    |   movel([0.360000, -1.280308, -2.635825, -0.796256, 1.570796, 1.930796],accel_mss,speed_ms,0,blend_radius_m)
    |   movel([0.360158, -1.281026, -2.635415, -0.795948, 1.570796, 1.930954],accel_mss,speed_ms,0,blend_radius_m)
    |   movel([0.360117, -1.282337, -2.634665, -0.795387, 1.570796, 1.930913],accel_mss,speed_ms,0,blend_radius_m)
    |   movel([0.359973, -1.283681, -2.633894, -0.794814, 1.570796, 1.930769],accel_mss,speed_ms,0,blend_radius_m)
    |   movel([0.359706, -1.284183, -2.633605, -0.794600, 1.570796, 1.930502],accel_mss,speed_ms,0,blend_radius_m)
    |   movel([0.359553, -1.284531, -2.633405, -0.794453, 1.570796, 1.930349],accel_mss,speed_ms,0,blend_radius_m)
    |   movel([0.359665, -1.284681, -2.633319, -0.794389, 1.570796, 1.930461],accel_mss,speed_ms,0,blend_radius_m)
    |   movel([0.360589, -1.285200, -2.633020, -0.794169, 1.570796, 1.931386],accel_mss,speed_ms,0,blend_radius_m)
    |   movel([0.360909, -1.283859, -2.633792, -0.794738, 1.570796, 1.931705],accel_mss,speed_ms,0,blend_radius_m)
    |   movel([0.361092, -1.281386, -2.635209, -0.795794, 1.570796, 1.931889],accel_mss,speed_ms,0,blend_radius_m)
    |   speed_ms = 0.005
    |   movel([0.361092, -1.272070, -2.630766, -0.809554, 1.570796, 1.931889],accel_mss,speed_ms,0,blend_radius_m)
    |   speed_ms = 0.040
    |   movel([0.352046, -1.270244, -2.631793, -0.810352, 1.570796, 1.922843],accel_mss,speed_ms,0,blend_radius_m)
    |   speed_ms = 0.005
    |   movel([0.352046, -1.279570, -2.636246, -0.796574, 1.570796, 1.922843],accel_mss,speed_ms,0,blend_radius_m)
    |   speed_ms = 0.025
    |   movel([0.350726, -1.280552, -2.635686, -0.796151, 1.570796, 1.921522],accel_mss,speed_ms,0,blend_radius_m)
    |   movel([0.350409, -1.280755, -2.635570, -0.796064, 1.570796, 1.921205],accel_mss,speed_ms,0,blend_radius_m)
    |   movel([0.349573, -1.281438, -2.635180, -0.795771, 1.570796, 1.920369],accel_mss,speed_ms,0,blend_radius_m)
    |   movel([0.349367, -1.281688, -2.635037, -0.795664, 1.570796, 1.920163],accel_mss,speed_ms,0,blend_radius_m)
    |   movel([0.349281, -1.282014, -2.634850, -0.795525, 1.570796, 1.920078],accel_mss,speed_ms,0,blend_radius_m)
    |   movel([0.349376, -1.282211, -2.634737, -0.795441, 1.570796, 1.920172],accel_mss,speed_ms,0,blend_radius_m)
    |   movel([0.349450, -1.282722, -2.634445, -0.795223, 1.570796, 1.920246],accel_mss,speed_ms,0,blend_radius_m)
    |   movel([0.349219, -1.283722, -2.633871, -0.794797, 1.570796, 1.920015],accel_mss,speed_ms,0,blend_radius_m)
    |   movel([0.348833, -1.284811, -2.633244, -0.794334, 1.570796, 1.919629],accel_mss,speed_ms,0,blend_radius_m)
    |   movel([0.348360, -1.285691, -2.632736, -0.793961, 1.570796, 1.919156],accel_mss,speed_ms,0,blend_radius_m)
    |   movel([0.346176, -1.288603, -2.631050, -0.792735, 1.570796, 1.916973],accel_mss,speed_ms,0,blend_radius_m)
    |   movel([0.345853, -1.288937, -2.630857, -0.792595, 1.570796, 1.916649],accel_mss,speed_ms,0,blend_radius_m)
    |   movel([0.345592, -1.289084, -2.630771, -0.792534, 1.570796, 1.916388],accel_mss,speed_ms,0,blend_radius_m)
    |   movel([0.345282, -1.289128, -2.630746, -0.792515, 1.570796, 1.916078],accel_mss,speed_ms,0,blend_radius_m)
    |   movel([0.344779, -1.289269, -2.630664, -0.792457, 1.570796, 1.915576],accel_mss,speed_ms,0,blend_radius_m)
    |   movel([0.344577, -1.289528, -2.630513, -0.792348, 1.570796, 1.915373],accel_mss,speed_ms,0,blend_radius_m)
    |   movel([0.343400, -1.291475, -2.629377, -0.791537, 1.570796, 1.914196],accel_mss,speed_ms,0,blend_radius_m)
    |   movel([0.342359, -1.292811, -2.628595, -0.790983, 1.570796, 1.913155],accel_mss,speed_ms,0,blend_radius_m)
    |   movel([0.341234, -1.294031, -2.627879, -0.790479, 1.570796, 1.912031],accel_mss,speed_ms,0,blend_radius_m)
    |   movel([0.340185, -1.294941, -2.627344, -0.790104, 1.570796, 1.910981],accel_mss,speed_ms,0,blend_radius_m)
    |   movel([0.339211, -1.295614, -2.626947, -0.789828, 1.570796, 1.910007],accel_mss,speed_ms,0,blend_radius_m)
    |   movel([0.338682, -1.295791, -2.626843, -0.789755, 1.570796, 1.909478],accel_mss,speed_ms,0,blend_radius_m)
    |   movel([0.338447, -1.295587, -2.626963, -0.789839, 1.570796, 1.909243],accel_mss,speed_ms,0,blend_radius_m)
    |   movel([0.338512, -1.294948, -2.627340, -0.790101, 1.570796, 1.909309],accel_mss,speed_ms,0,blend_radius_m)
    |   movel([0.338713, -1.294120, -2.627827, -0.790442, 1.570796, 1.909510],accel_mss,speed_ms,0,blend_radius_m)
    |   movel([0.338129, -1.294814, -2.627419, -0.790156, 1.570796, 1.908925],accel_mss,speed_ms,0,blend_radius_m)
    |   movel([0.335286, -1.297812, -2.625648, -0.788929, 1.570796, 1.906082],accel_mss,speed_ms,0,blend_radius_m)
    |   movel([0.333596, -1.299421, -2.624693, -0.788275, 1.570796, 1.904392],accel_mss,speed_ms,0,blend_radius_m)
    |   movel([0.330932, -1.301652, -2.623363, -0.787375, 1.570796, 1.901728],accel_mss,speed_ms,0,blend_radius_m)
    |   movel([0.330138, -1.302174, -2.623051, -0.787165, 1.570796, 1.900934],accel_mss,speed_ms,0,blend_radius_m)
    |   movel([0.329651, -1.302339, -2.622952, -0.787098, 1.570796, 1.900448],accel_mss,speed_ms,0,blend_radius_m)
    |   movel([0.329404, -1.302208, -2.623030, -0.787151, 1.570796, 1.900200],accel_mss,speed_ms,0,blend_radius_m)
    |   movel([0.329712, -1.301575, -2.623409, -0.787406, 1.570796, 1.900508],accel_mss,speed_ms,0,blend_radius_m)
    |   movel([0.330081, -1.300968, -2.623771, -0.787650, 1.570796, 1.900877],accel_mss,speed_ms,0,blend_radius_m)
    |   movel([0.331306, -1.299082, -2.624894, -0.788413, 1.570796, 1.902102],accel_mss,speed_ms,0,blend_radius_m)
    |   movel([0.331670, -1.298377, -2.625312, -0.788699, 1.570796, 1.902467],accel_mss,speed_ms,0,blend_radius_m)
    |   movel([0.332580, -1.295268, -2.627151, -0.789970, 1.570796, 1.903377],accel_mss,speed_ms,0,blend_radius_m)
    |   movel([0.332687, -1.295094, -2.627254, -0.790041, 1.570796, 1.903483],accel_mss,speed_ms,0,blend_radius_m)
    |   movel([0.333051, -1.294898, -2.627369, -0.790122, 1.570796, 1.903847],accel_mss,speed_ms,0,blend_radius_m)
    |   movel([0.333400, -1.294997, -2.627311, -0.790081, 1.570796, 1.904196],accel_mss,speed_ms,0,blend_radius_m)
    |   movel([0.333513, -1.295473, -2.627031, -0.789886, 1.570796, 1.904310],accel_mss,speed_ms,0,blend_radius_m)
    |   movel([0.333369, -1.296352, -2.626512, -0.789526, 1.570796, 1.904165],accel_mss,speed_ms,0,blend_radius_m)
    |   movel([0.332468, -1.299246, -2.624796, -0.788346, 1.570796, 1.903264],accel_mss,speed_ms,0,blend_radius_m)
    |   movel([0.333060, -1.298841, -2.625038, -0.788511, 1.570796, 1.903857],accel_mss,speed_ms,0,blend_radius_m)
    |   movel([0.334701, -1.297178, -2.626023, -0.789188, 1.570796, 1.905498],accel_mss,speed_ms,0,blend_radius_m)
    |   movel([0.339129, -1.292381, -2.628847, -0.791161, 1.570796, 1.909925],accel_mss,speed_ms,0,blend_radius_m)
    |   movel([0.339470, -1.292099, -2.629012, -0.791278, 1.570796, 1.910266],accel_mss,speed_ms,0,blend_radius_m)
    |   movel([0.339852, -1.291915, -2.629120, -0.791354, 1.570796, 1.910648],accel_mss,speed_ms,0,blend_radius_m)
    |   movel([0.340105, -1.291922, -2.629116, -0.791351, 1.570796, 1.910901],accel_mss,speed_ms,0,blend_radius_m)
    |   movel([0.340213, -1.292101, -2.629011, -0.791277, 1.570796, 1.911009],accel_mss,speed_ms,0,blend_radius_m)
    |   movel([0.340131, -1.293204, -2.628365, -0.790820, 1.570796, 1.910927],accel_mss,speed_ms,0,blend_radius_m)
    |   movel([0.340095, -1.293842, -2.627990, -0.790557, 1.570796, 1.910891],accel_mss,speed_ms,0,blend_radius_m)
    |   movel([0.340385, -1.293737, -2.628052, -0.790600, 1.570796, 1.911181],accel_mss,speed_ms,0,blend_radius_m)
    |   movel([0.341029, -1.293046, -2.628457, -0.790885, 1.570796, 1.911825],accel_mss,speed_ms,0,blend_radius_m)
    |   movel([0.342320, -1.291451, -2.629392, -0.791547, 1.570796, 1.913117],accel_mss,speed_ms,0,blend_radius_m)
    |   movel([0.342678, -1.290913, -2.629706, -0.791771, 1.570796, 1.913474],accel_mss,speed_ms,0,blend_radius_m)
    |   movel([0.344707, -1.287200, -2.631864, -0.793325, 1.570796, 1.915504],accel_mss,speed_ms,0,blend_radius_m)
    |   movel([0.345022, -1.286686, -2.632162, -0.793541, 1.570796, 1.915819],accel_mss,speed_ms,0,blend_radius_m)
    |   movel([0.345276, -1.286420, -2.632316, -0.793654, 1.570796, 1.916072],accel_mss,speed_ms,0,blend_radius_m)
    |   movel([0.345565, -1.286274, -2.632400, -0.793715, 1.570796, 1.916361],accel_mss,speed_ms,0,blend_radius_m)
    |   movel([0.345919, -1.286308, -2.632380, -0.793701, 1.570796, 1.916715],accel_mss,speed_ms,0,blend_radius_m)
    |   movel([0.345989, -1.286458, -2.632294, -0.793638, 1.570796, 1.916786],accel_mss,speed_ms,0,blend_radius_m)
    |   movel([0.346060, -1.287092, -2.631927, -0.793370, 1.570796, 1.916857],accel_mss,speed_ms,0,blend_radius_m)
    |   movel([0.346199, -1.287137, -2.631901, -0.793351, 1.570796, 1.916995],accel_mss,speed_ms,0,blend_radius_m)
    |   movel([0.346613, -1.286673, -2.632169, -0.793547, 1.570796, 1.917409],accel_mss,speed_ms,0,blend_radius_m)
    |   movel([0.347721, -1.284766, -2.633270, -0.794353, 1.570796, 1.918517],accel_mss,speed_ms,0,blend_radius_m)
    |   movel([0.348015, -1.284034, -2.633691, -0.794664, 1.570796, 1.918811],accel_mss,speed_ms,0,blend_radius_m)
    |   movel([0.348173, -1.283275, -2.634127, -0.794987, 1.570796, 1.918969],accel_mss,speed_ms,0,blend_radius_m)
    |   movel([0.348061, -1.283203, -2.634169, -0.795018, 1.570796, 1.918858],accel_mss,speed_ms,0,blend_radius_m)
    |   movel([0.347358, -1.283201, -2.634170, -0.795018, 1.570796, 1.918154],accel_mss,speed_ms,0,blend_radius_m)
    |   movel([0.347299, -1.282914, -2.634334, -0.795141, 1.570796, 1.918095],accel_mss,speed_ms,0,blend_radius_m)
    |   movel([0.347686, -1.282282, -2.634697, -0.795411, 1.570796, 1.918482],accel_mss,speed_ms,0,blend_radius_m)
    |   movel([0.348658, -1.281144, -2.635348, -0.795897, 1.570796, 1.919454],accel_mss,speed_ms,0,blend_radius_m)
    |   movel([0.350016, -1.279729, -2.636155, -0.796505, 1.570796, 1.920812],accel_mss,speed_ms,0,blend_radius_m)
    |   movel([0.350378, -1.279523, -2.636273, -0.796594, 1.570796, 1.921174],accel_mss,speed_ms,0,blend_radius_m)
    |   movel([0.351006, -1.279344, -2.636374, -0.796671, 1.570796, 1.921802],accel_mss,speed_ms,0,blend_radius_m)
    |   movel([0.351161, -1.279219, -2.636445, -0.796725, 1.570796, 1.921958],accel_mss,speed_ms,0,blend_radius_m)
    |   movel([0.351485, -1.278767, -2.636702, -0.796920, 1.570796, 1.922281],accel_mss,speed_ms,0,blend_radius_m)
    |   movel([0.351478, -1.278534, -2.636835, -0.797020, 1.570796, 1.922274],accel_mss,speed_ms,0,blend_radius_m)
    |   movel([0.350699, -1.278105, -2.637078, -0.797206, 1.570796, 1.921496],accel_mss,speed_ms,0,blend_radius_m)
    |   movel([0.350151, -1.277985, -2.637146, -0.797258, 1.570796, 1.920947],accel_mss,speed_ms,0,blend_radius_m)
    |   movel([0.348867, -1.278148, -2.637054, -0.797187, 1.570796, 1.919663],accel_mss,speed_ms,0,blend_radius_m)
    |   movel([0.348187, -1.278424, -2.636897, -0.797068, 1.570796, 1.918984],accel_mss,speed_ms,0,blend_radius_m)
    |   movel([0.346556, -1.279452, -2.636312, -0.796624, 1.570796, 1.917352],accel_mss,speed_ms,0,blend_radius_m)
    |   movel([0.344489, -1.281187, -2.635323, -0.795879, 1.570796, 1.915285],accel_mss,speed_ms,0,blend_radius_m)
    |   movel([0.342140, -1.283410, -2.634050, -0.794929, 1.570796, 1.912937],accel_mss,speed_ms,0,blend_radius_m)
    |   movel([0.339990, -1.285647, -2.632762, -0.793980, 1.570796, 1.910786],accel_mss,speed_ms,0,blend_radius_m)
    |   movel([0.338281, -1.287605, -2.631630, -0.793154, 1.570796, 1.909077],accel_mss,speed_ms,0,blend_radius_m)
    |   movel([0.337925, -1.288106, -2.631339, -0.792944, 1.570796, 1.908722],accel_mss,speed_ms,0,blend_radius_m)
    |   movel([0.337295, -1.289450, -2.630558, -0.792381, 1.570796, 1.908092],accel_mss,speed_ms,0,blend_radius_m)
    |   movel([0.336751, -1.290223, -2.630108, -0.792058, 1.570796, 1.907547],accel_mss,speed_ms,0,blend_radius_m)
    |   movel([0.335966, -1.291041, -2.629631, -0.791717, 1.570796, 1.906762],accel_mss,speed_ms,0,blend_radius_m)
    |   movel([0.334835, -1.292017, -2.629060, -0.791312, 1.570796, 1.905631],accel_mss,speed_ms,0,blend_radius_m)
    |   movel([0.333094, -1.293432, -2.628231, -0.790726, 1.570796, 1.903890],accel_mss,speed_ms,0,blend_radius_m)
    |   movel([0.333989, -1.293324, -2.628294, -0.790771, 1.570796, 1.904785],accel_mss,speed_ms,0,blend_radius_m)
    |   movel([0.334947, -1.293151, -2.628396, -0.790842, 1.570796, 1.905743],accel_mss,speed_ms,0,blend_radius_m)
    |   movel([0.335825, -1.292864, -2.628564, -0.790961, 1.570796, 1.906621],accel_mss,speed_ms,0,blend_radius_m)
    |   movel([0.336611, -1.292469, -2.628796, -0.791124, 1.570796, 1.907408],accel_mss,speed_ms,0,blend_radius_m)
    |   movel([0.337314, -1.291964, -2.629091, -0.791334, 1.570796, 1.908110],accel_mss,speed_ms,0,blend_radius_m)
    |   movel([0.339476, -1.289654, -2.630440, -0.792296, 1.570796, 1.910272],accel_mss,speed_ms,0,blend_radius_m)
    |   movel([0.340428, -1.288554, -2.631079, -0.792756, 1.570796, 1.911224],accel_mss,speed_ms,0,blend_radius_m)
    |   movel([0.342358, -1.286351, -2.632355, -0.793683, 1.570796, 1.913154],accel_mss,speed_ms,0,blend_radius_m)
    |   movel([0.343884, -1.284770, -2.633268, -0.794351, 1.570796, 1.914681],accel_mss,speed_ms,0,blend_radius_m)
    |   movel([0.345057, -1.283720, -2.633872, -0.794798, 1.570796, 1.915853],accel_mss,speed_ms,0,blend_radius_m)
    |   movel([0.345391, -1.283506, -2.633994, -0.794888, 1.570796, 1.916188],accel_mss,speed_ms,0,blend_radius_m)
    |   movel([0.345733, -1.283407, -2.634051, -0.794931, 1.570796, 1.916529],accel_mss,speed_ms,0,blend_radius_m)
    |   movel([0.346062, -1.283485, -2.634007, -0.794897, 1.570796, 1.916858],accel_mss,speed_ms,0,blend_radius_m)
    |   movel([0.346078, -1.283751, -2.633854, -0.794784, 1.570796, 1.916875],accel_mss,speed_ms,0,blend_radius_m)
    |   movel([0.345707, -1.284258, -2.633562, -0.794569, 1.570796, 1.916503],accel_mss,speed_ms,0,blend_radius_m)
    |   movel([0.343367, -1.286602, -2.632210, -0.793577, 1.570796, 1.914163],accel_mss,speed_ms,0,blend_radius_m)
    |   movel([0.342356, -1.287721, -2.631562, -0.793106, 1.570796, 1.913152],accel_mss,speed_ms,0,blend_radius_m)
    |   movel([0.339475, -1.291018, -2.629644, -0.791727, 1.570796, 1.910271],accel_mss,speed_ms,0,blend_radius_m)
    |   movel([0.338056, -1.292411, -2.628830, -0.791148, 1.570796, 1.908853],accel_mss,speed_ms,0,blend_radius_m)
    |   movel([0.336846, -1.293317, -2.628299, -0.790774, 1.570796, 1.907642],accel_mss,speed_ms,0,blend_radius_m)
    |   movel([0.335632, -1.293912, -2.627949, -0.790528, 1.570796, 1.906428],accel_mss,speed_ms,0,blend_radius_m)
    |   movel([0.332841, -1.294566, -2.627564, -0.790258, 1.570796, 1.903637],accel_mss,speed_ms,0,blend_radius_m)
    |   movel([0.331679, -1.294769, -2.627445, -0.790175, 1.570796, 1.902475],accel_mss,speed_ms,0,blend_radius_m)
    |   movel([0.329311, -1.295109, -2.627245, -0.790035, 1.570796, 1.900107],accel_mss,speed_ms,0,blend_radius_m)
    |   movel([0.328965, -1.295079, -2.627263, -0.790048, 1.570796, 1.899762],accel_mss,speed_ms,0,blend_radius_m)
    |   movel([0.328847, -1.294931, -2.627350, -0.790108, 1.570796, 1.899643],accel_mss,speed_ms,0,blend_radius_m)
    |   movel([0.328941, -1.294638, -2.627522, -0.790229, 1.570796, 1.899737],accel_mss,speed_ms,0,blend_radius_m)
    |   movel([0.329215, -1.294351, -2.627691, -0.790347, 1.570796, 1.900011],accel_mss,speed_ms,0,blend_radius_m)
    |   movel([0.329727, -1.294034, -2.627877, -0.790478, 1.570796, 1.900523],accel_mss,speed_ms,0,blend_radius_m)
    |   movel([0.331665, -1.293098, -2.628427, -0.790864, 1.570796, 1.902462],accel_mss,speed_ms,0,blend_radius_m)
    |   movel([0.332996, -1.292293, -2.628899, -0.791197, 1.570796, 1.903793],accel_mss,speed_ms,0,blend_radius_m)
    |   movel([0.334270, -1.291420, -2.629410, -0.791560, 1.570796, 1.905066],accel_mss,speed_ms,0,blend_radius_m)
    |   movel([0.335177, -1.290667, -2.629849, -0.791873, 1.570796, 1.905974],accel_mss,speed_ms,0,blend_radius_m)
    |   movel([0.335919, -1.289820, -2.630343, -0.792226, 1.570796, 1.906715],accel_mss,speed_ms,0,blend_radius_m)
    |   movel([0.336246, -1.289316, -2.630636, -0.792437, 1.570796, 1.907043],accel_mss,speed_ms,0,blend_radius_m)
    |   movel([0.337469, -1.287167, -2.631884, -0.793339, 1.570796, 1.908266],accel_mss,speed_ms,0,blend_radius_m)
    |   movel([0.337607, -1.286986, -2.631988, -0.793415, 1.570796, 1.908403],accel_mss,speed_ms,0,blend_radius_m)
    |   movel([0.337528, -1.286900, -2.632038, -0.793451, 1.570796, 1.908324],accel_mss,speed_ms,0,blend_radius_m)
    |   movel([0.337263, -1.286966, -2.632000, -0.793423, 1.570796, 1.908059],accel_mss,speed_ms,0,blend_radius_m)
    |   movel([0.336794, -1.286946, -2.632011, -0.793432, 1.570796, 1.907591],accel_mss,speed_ms,0,blend_radius_m)
    |   movel([0.336758, -1.286839, -2.632073, -0.793477, 1.570796, 1.907555],accel_mss,speed_ms,0,blend_radius_m)
    |   movel([0.336882, -1.286488, -2.632276, -0.793625, 1.570796, 1.907678],accel_mss,speed_ms,0,blend_radius_m)
    |   movel([0.337579, -1.285557, -2.632814, -0.794018, 1.570796, 1.908376],accel_mss,speed_ms,0,blend_radius_m)
    |   movel([0.340525, -1.282052, -2.634828, -0.795509, 1.570796, 1.911322],accel_mss,speed_ms,0,blend_radius_m)
    |   movel([0.340661, -1.281806, -2.634969, -0.795614, 1.570796, 1.911457],accel_mss,speed_ms,0,blend_radius_m)
    |   movel([0.340523, -1.281433, -2.635183, -0.795774, 1.570796, 1.911319],accel_mss,speed_ms,0,blend_radius_m)
    |   movel([0.340591, -1.280649, -2.635631, -0.796110, 1.570796, 1.911388],accel_mss,speed_ms,0,blend_radius_m)
    |   movel([0.340729, -1.279843, -2.636090, -0.796456, 1.570796, 1.911526],accel_mss,speed_ms,0,blend_radius_m)
    |   movel([0.340926, -1.279484, -2.636294, -0.796610, 1.570796, 1.911722],accel_mss,speed_ms,0,blend_radius_m)
    |   movel([0.341239, -1.279281, -2.636410, -0.796698, 1.570796, 1.912035],accel_mss,speed_ms,0,blend_radius_m)
    |   movel([0.341530, -1.279306, -2.636396, -0.796687, 1.570796, 1.912326],accel_mss,speed_ms,0,blend_radius_m)
    |   movel([0.341737, -1.279581, -2.636239, -0.796569, 1.570796, 1.912533],accel_mss,speed_ms,0,blend_radius_m)
    |   movel([0.341803, -1.280049, -2.635973, -0.796368, 1.570796, 1.912599],accel_mss,speed_ms,0,blend_radius_m)
    |   movel([0.341795, -1.280796, -2.635547, -0.796047, 1.570796, 1.912592],accel_mss,speed_ms,0,blend_radius_m)
    |   movel([0.343174, -1.279535, -2.636265, -0.796588, 1.570796, 1.913971],accel_mss,speed_ms,0,blend_radius_m)
    |   movel([0.346049, -1.276916, -2.637752, -0.797721, 1.570796, 1.916846],accel_mss,speed_ms,0,blend_radius_m)
    |   movel([0.345679, -1.276653, -2.637901, -0.797835, 1.570796, 1.916476],accel_mss,speed_ms,0,blend_radius_m)
    |   movel([0.345163, -1.276545, -2.637962, -0.797882, 1.570796, 1.915960],accel_mss,speed_ms,0,blend_radius_m)
    |   movel([0.344787, -1.276712, -2.637868, -0.797809, 1.570796, 1.915584],accel_mss,speed_ms,0,blend_radius_m)
    |   movel([0.341919, -1.278507, -2.636850, -0.797032, 1.570796, 1.912716],accel_mss,speed_ms,0,blend_radius_m)
    |   movel([0.340652, -1.279583, -2.636238, -0.796568, 1.570796, 1.911449],accel_mss,speed_ms,0,blend_radius_m)
    |   movel([0.339694, -1.280798, -2.635545, -0.796046, 1.570796, 1.910490],accel_mss,speed_ms,0,blend_radius_m)
    |   movel([0.338762, -1.282492, -2.634576, -0.795321, 1.570796, 1.909558],accel_mss,speed_ms,0,blend_radius_m)
    |   movel([0.337668, -1.284650, -2.633337, -0.794402, 1.570796, 1.908464],accel_mss,speed_ms,0,blend_radius_m)
    |   movel([0.337414, -1.284913, -2.633185, -0.794291, 1.570796, 1.908211],accel_mss,speed_ms,0,blend_radius_m)
    |   movel([0.337121, -1.285037, -2.633114, -0.794238, 1.570796, 1.907917],accel_mss,speed_ms,0,blend_radius_m)
    |   movel([0.336837, -1.284954, -2.633162, -0.794273, 1.570796, 1.907633],accel_mss,speed_ms,0,blend_radius_m)
    |   movel([0.336775, -1.284660, -2.633331, -0.794398, 1.570796, 1.907571],accel_mss,speed_ms,0,blend_radius_m)
    |   movel([0.336965, -1.284046, -2.633684, -0.794659, 1.570796, 1.907762],accel_mss,speed_ms,0,blend_radius_m)
    |   movel([0.338700, -1.280649, -2.635630, -0.796110, 1.570796, 1.909496],accel_mss,speed_ms,0,blend_radius_m)
    |   movel([0.339219, -1.279877, -2.636071, -0.796441, 1.570796, 1.910015],accel_mss,speed_ms,0,blend_radius_m)
    |   movel([0.340505, -1.278475, -2.636868, -0.797046, 1.570796, 1.911301],accel_mss,speed_ms,0,blend_radius_m)
    |   movel([0.341242, -1.277887, -2.637202, -0.797300, 1.570796, 1.912038],accel_mss,speed_ms,0,blend_radius_m)
    |   movel([0.344850, -1.275621, -2.638484, -0.798284, 1.570796, 1.915646],accel_mss,speed_ms,0,blend_radius_m)
    |   movel([0.344975, -1.275480, -2.638564, -0.798345, 1.570796, 1.915771],accel_mss,speed_ms,0,blend_radius_m)
    |   movel([0.344967, -1.275345, -2.638640, -0.798404, 1.570796, 1.915763],accel_mss,speed_ms,0,blend_radius_m)
    |   movel([0.344595, -1.275334, -2.638646, -0.798409, 1.570796, 1.915392],accel_mss,speed_ms,0,blend_radius_m)
    |   movel([0.342920, -1.276167, -2.638176, -0.798046, 1.570796, 1.913716],accel_mss,speed_ms,0,blend_radius_m)
    |   movel([0.340911, -1.277359, -2.637501, -0.797528, 1.570796, 1.911707],accel_mss,speed_ms,0,blend_radius_m)
    |   movel([0.340160, -1.277929, -2.637178, -0.797282, 1.570796, 1.910956],accel_mss,speed_ms,0,blend_radius_m)
    |   movel([0.339476, -1.278577, -2.636810, -0.797002, 1.570796, 1.910272],accel_mss,speed_ms,0,blend_radius_m)
    |   movel([0.338291, -1.280119, -2.635933, -0.796337, 1.570796, 1.909087],accel_mss,speed_ms,0,blend_radius_m)
    |   movel([0.337053, -1.282368, -2.634647, -0.795373, 1.570796, 1.907849],accel_mss,speed_ms,0,blend_radius_m)
    |   movel([0.335830, -1.284771, -2.633267, -0.794351, 1.570796, 1.906627],accel_mss,speed_ms,0,blend_radius_m)
    |   movel([0.335570, -1.285106, -2.633074, -0.794209, 1.570796, 1.906366],accel_mss,speed_ms,0,blend_radius_m)
    |   movel([0.335251, -1.285332, -2.632944, -0.794113, 1.570796, 1.906047],accel_mss,speed_ms,0,blend_radius_m)
    |   movel([0.334956, -1.285396, -2.632907, -0.794086, 1.570796, 1.905752],accel_mss,speed_ms,0,blend_radius_m)
    |   movel([0.334753, -1.285283, -2.632972, -0.794134, 1.570796, 1.905550],accel_mss,speed_ms,0,blend_radius_m)
    |   movel([0.334737, -1.285068, -2.633096, -0.794225, 1.570796, 1.905533],accel_mss,speed_ms,0,blend_radius_m)
    |   movel([0.335255, -1.283844, -2.633800, -0.794745, 1.570796, 1.906051],accel_mss,speed_ms,0,blend_radius_m)
    |   movel([0.335912, -1.282552, -2.634542, -0.795295, 1.570796, 1.906709],accel_mss,speed_ms,0,blend_radius_m)
    |   movel([0.337597, -1.279500, -2.636285, -0.796603, 1.570796, 1.908393],accel_mss,speed_ms,0,blend_radius_m)
    |   movel([0.338195, -1.278676, -2.636754, -0.796959, 1.570796, 1.908991],accel_mss,speed_ms,0,blend_radius_m)
    |   movel([0.339703, -1.277153, -2.637618, -0.797618, 1.570796, 1.910499],accel_mss,speed_ms,0,blend_radius_m)
    |   movel([0.340471, -1.276557, -2.637955, -0.797876, 1.570796, 1.911267],accel_mss,speed_ms,0,blend_radius_m)
    |   movel([0.342715, -1.275234, -2.638703, -0.798452, 1.570796, 1.913511],accel_mss,speed_ms,0,blend_radius_m)
    |   movel([0.344071, -1.274571, -2.639076, -0.798742, 1.570796, 1.914867],accel_mss,speed_ms,0,blend_radius_m)
    |   movel([0.345029, -1.274259, -2.639252, -0.798878, 1.570796, 1.915825],accel_mss,speed_ms,0,blend_radius_m)
    |   movel([0.345612, -1.274279, -2.639241, -0.798869, 1.570796, 1.916408],accel_mss,speed_ms,0,blend_radius_m)
    |   movel([0.346261, -1.275264, -2.638686, -0.798439, 1.570796, 1.917057],accel_mss,speed_ms,0,blend_radius_m)
    |   movel([0.346498, -1.275497, -2.638554, -0.798338, 1.570796, 1.917295],accel_mss,speed_ms,0,blend_radius_m)
    |   movel([0.347072, -1.275880, -2.638338, -0.798171, 1.570796, 1.917869],accel_mss,speed_ms,0,blend_radius_m)
    |   movel([0.347297, -1.275882, -2.638337, -0.798170, 1.570796, 1.918094],accel_mss,speed_ms,0,blend_radius_m)
    |   movel([0.348230, -1.275526, -2.638538, -0.798325, 1.570796, 1.919027],accel_mss,speed_ms,0,blend_radius_m)
    |   movel([0.348990, -1.275437, -2.638588, -0.798364, 1.570796, 1.919786],accel_mss,speed_ms,0,blend_radius_m)
    |   movel([0.349669, -1.275526, -2.638538, -0.798325, 1.570796, 1.920466],accel_mss,speed_ms,0,blend_radius_m)
    |   movel([0.350116, -1.275789, -2.638390, -0.798211, 1.570796, 1.920912],accel_mss,speed_ms,0,blend_radius_m)
    |   movel([0.350438, -1.276356, -2.638069, -0.797964, 1.570796, 1.921235],accel_mss,speed_ms,0,blend_radius_m)
    |   movel([0.350427, -1.276487, -2.637995, -0.797907, 1.570796, 1.921223],accel_mss,speed_ms,0,blend_radius_m)
    |   movel([0.350632, -1.276776, -2.637832, -0.797782, 1.570796, 1.921429],accel_mss,speed_ms,0,blend_radius_m)
    |   movel([0.350810, -1.276823, -2.637805, -0.797761, 1.570796, 1.921606],accel_mss,speed_ms,0,blend_radius_m)
    |   movel([0.351648, -1.277063, -2.637669, -0.797657, 1.570796, 1.922445],accel_mss,speed_ms,0,blend_radius_m)
    |   movel([0.352340, -1.277521, -2.637409, -0.797458, 1.570796, 1.923136],accel_mss,speed_ms,0,blend_radius_m)
    |   movel([0.352766, -1.278081, -2.637092, -0.797216, 1.570796, 1.923562],accel_mss,speed_ms,0,blend_radius_m)
    |   movel([0.352762, -1.278621, -2.636785, -0.796983, 1.570796, 1.923559],accel_mss,speed_ms,0,blend_radius_m)
    |   movel([0.352273, -1.279335, -2.636379, -0.796675, 1.570796, 1.923069],accel_mss,speed_ms,0,blend_radius_m)
    |   movel([0.352046, -1.279570, -2.636246, -0.796574, 1.570796, 1.922843],accel_mss,speed_ms,0,blend_radius_m)
    |   movel([0.350726, -1.280552, -2.635686, -0.796151, 1.570796, 1.921522],accel_mss,speed_ms,0,blend_radius_m)
    |   movel([0.350409, -1.280755, -2.635570, -0.796064, 1.570796, 1.921205],accel_mss,speed_ms,0,blend_radius_m)
    |   movel([0.349573, -1.281438, -2.635180, -0.795771, 1.570796, 1.920369],accel_mss,speed_ms,0,blend_radius_m)
    |   movel([0.349449, -1.281590, -2.635093, -0.795706, 1.570796, 1.920245],accel_mss,speed_ms,0,blend_radius_m)
    |   speed_ms = 0.005
    |   movel([0.349449, -1.272274, -2.630650, -0.809465, 1.570796, 1.920245],accel_mss,speed_ms,0,blend_radius_m)
    |   speed_ms = 0.040
    |   movel([0.349144, -1.267306, -2.633439, -0.811644, 1.570796, 1.919941],accel_mss,speed_ms,0,blend_radius_m)
    |   speed_ms = 0.005
    |   movel([0.349144, -1.276648, -2.637904, -0.797837, 1.570796, 1.919941],accel_mss,speed_ms,0,blend_radius_m)
    |   speed_ms = 0.025
    |   movel([0.349180, -1.276811, -2.637812, -0.797766, 1.570796, 1.919976],accel_mss,speed_ms,0,blend_radius_m)
    |   movel([0.349084, -1.276963, -2.637725, -0.797700, 1.570796, 1.919880],accel_mss,speed_ms,0,blend_radius_m)
    |   movel([0.348249, -1.277348, -2.637508, -0.797533, 1.570796, 1.919045],accel_mss,speed_ms,0,blend_radius_m)
    |   movel([0.347099, -1.277982, -2.637148, -0.797259, 1.570796, 1.917896],accel_mss,speed_ms,0,blend_radius_m)
    |   movel([0.345154, -1.279499, -2.636286, -0.796604, 1.570796, 1.915950],accel_mss,speed_ms,0,blend_radius_m)
    |   movel([0.343016, -1.281354, -2.635228, -0.795807, 1.570796, 1.913812],accel_mss,speed_ms,0,blend_radius_m)
    |   movel([0.339384, -1.284965, -2.633155, -0.794269, 1.570796, 1.910180],accel_mss,speed_ms,0,blend_radius_m)
    |   movel([0.338860, -1.285472, -2.632863, -0.794054, 1.570796, 1.909657],accel_mss,speed_ms,0,blend_radius_m)
    |   movel([0.339303, -1.284870, -2.633210, -0.794309, 1.570796, 1.910099],accel_mss,speed_ms,0,blend_radius_m)
    |   movel([0.341971, -1.281947, -2.634889, -0.795554, 1.570796, 1.912767],accel_mss,speed_ms,0,blend_radius_m)
    |   movel([0.343425, -1.280525, -2.635701, -0.796163, 1.570796, 1.914221],accel_mss,speed_ms,0,blend_radius_m)
    |   movel([0.346674, -1.277583, -2.637374, -0.797432, 1.570796, 1.917470],accel_mss,speed_ms,0,blend_radius_m)
    |   movel([0.347380, -1.277019, -2.637694, -0.797676, 1.570796, 1.918176],accel_mss,speed_ms,0,blend_radius_m)
    |   movel([0.347867, -1.276745, -2.637849, -0.797795, 1.570796, 1.918663],accel_mss,speed_ms,0,blend_radius_m)
    |   movel([0.348359, -1.276612, -2.637924, -0.797853, 1.570796, 1.919155],accel_mss,speed_ms,0,blend_radius_m)
    |   movel([0.349144, -1.276648, -2.637904, -0.797837, 1.570796, 1.919941],accel_mss,speed_ms,0,blend_radius_m)
    |   movel([0.349180, -1.276811, -2.637812, -0.797766, 1.570796, 1.919976],accel_mss,speed_ms,0,blend_radius_m)
    |   movel([0.349084, -1.276963, -2.637725, -0.797700, 1.570796, 1.919880],accel_mss,speed_ms,0,blend_radius_m)
    |   movel([0.348249, -1.277348, -2.637508, -0.797533, 1.570796, 1.919045],accel_mss,speed_ms,0,blend_radius_m)
    |   movel([0.347099, -1.277982, -2.637148, -0.797259, 1.570796, 1.917896],accel_mss,speed_ms,0,blend_radius_m)
    |   movel([0.346664, -1.278321, -2.636955, -0.797112, 1.570796, 1.917460],accel_mss,speed_ms,0,blend_radius_m)
    |   speed_ms = 0.005
    |   movel([0.346664, -1.268989, -2.632498, -0.810902, 1.570796, 1.917460],accel_mss,speed_ms,0,blend_radius_m)
    |   speed_ms = 0.040
    |   movel([0.355687, -1.252153, -2.641759, -0.818477, 1.570796, 1.926483],accel_mss,speed_ms,0,blend_radius_m)
    |   speed_ms = 0.005
    |   movel([0.355687, -1.261571, -2.646293, -0.804525, 1.570796, 1.926483],accel_mss,speed_ms,0,blend_radius_m)
    |   speed_ms = 0.025
    |   movel([0.352923, -1.261989, -2.646064, -0.804336, 1.570796, 1.923720],accel_mss,speed_ms,0,blend_radius_m)
    |   movel([0.351477, -1.262150, -2.645976, -0.804263, 1.570796, 1.922274],accel_mss,speed_ms,0,blend_radius_m)
    |   movel([0.347382, -1.262736, -2.645654, -0.803999, 1.570796, 1.918179],accel_mss,speed_ms,0,blend_radius_m)
    |   movel([0.346630, -1.262953, -2.645535, -0.803900, 1.570796, 1.917427],accel_mss,speed_ms,0,blend_radius_m)
    |   movel([0.345461, -1.263364, -2.645310, -0.803715, 1.570796, 1.916257],accel_mss,speed_ms,0,blend_radius_m)
    |   movel([0.346577, -1.263102, -2.645454, -0.803834, 1.570796, 1.917374],accel_mss,speed_ms,0,blend_radius_m)
    |   movel([0.348966, -1.262703, -2.645673, -0.804014, 1.570796, 1.919763],accel_mss,speed_ms,0,blend_radius_m)
    |   movel([0.350464, -1.262562, -2.645750, -0.804077, 1.570796, 1.921261],accel_mss,speed_ms,0,blend_radius_m)
    |   movel([0.354195, -1.262290, -2.645899, -0.804200, 1.570796, 1.924992],accel_mss,speed_ms,0,blend_radius_m)
    |   movel([0.354710, -1.262136, -2.645983, -0.804270, 1.570796, 1.925506],accel_mss,speed_ms,0,blend_radius_m)
    |   movel([0.355799, -1.261571, -2.646292, -0.804525, 1.570796, 1.926595],accel_mss,speed_ms,0,blend_radius_m)
    |   movel([0.353049, -1.261972, -2.646073, -0.804344, 1.570796, 1.923846],accel_mss,speed_ms,0,blend_radius_m)
    |   speed_ms = 0.005
    |   movel([0.353049, -1.252556, -2.641541, -0.818292, 1.570796, 1.923846],accel_mss,speed_ms,0,blend_radius_m)
    |   speed_ms = 0.040
    |   movel([0.364668, -1.244388, -2.645916, -0.822086, 1.570796, 1.935465],accel_mss,speed_ms,0,blend_radius_m)
    |   speed_ms = 0.005
    |   movel([0.364668, -1.253843, -2.650485, -0.808062, 1.570796, 1.935465],accel_mss,speed_ms,0,blend_radius_m)
    |   speed_ms = 0.025
    |   movel([0.363454, -1.255161, -2.649775, -0.807453, 1.570796, 1.934250],accel_mss,speed_ms,0,blend_radius_m)
    |   movel([0.362093, -1.256330, -2.649143, -0.806916, 1.570796, 1.932889],accel_mss,speed_ms,0,blend_radius_m)
    |   movel([0.360626, -1.257318, -2.648608, -0.806462, 1.570796, 1.931422],accel_mss,speed_ms,0,blend_radius_m)
    |   movel([0.359109, -1.258086, -2.648192, -0.806111, 1.570796, 1.929905],accel_mss,speed_ms,0,blend_radius_m)
    |   movel([0.357635, -1.258592, -2.647917, -0.805880, 1.570796, 1.928432],accel_mss,speed_ms,0,blend_radius_m)
    |   movel([0.356218, -1.258833, -2.647786, -0.805770, 1.570796, 1.927014],accel_mss,speed_ms,0,blend_radius_m)
    |   movel([0.354966, -1.258787, -2.647811, -0.805791, 1.570796, 1.925763],accel_mss,speed_ms,0,blend_radius_m)
    |   movel([0.353888, -1.258449, -2.647995, -0.805945, 1.570796, 1.924685],accel_mss,speed_ms,0,blend_radius_m)
    |   movel([0.353277, -1.258091, -2.648189, -0.806109, 1.570796, 1.924073],accel_mss,speed_ms,0,blend_radius_m)
    |   movel([0.353111, -1.257777, -2.648360, -0.806252, 1.570796, 1.923908],accel_mss,speed_ms,0,blend_radius_m)
    |   movel([0.353257, -1.257383, -2.648573, -0.806433, 1.570796, 1.924053],accel_mss,speed_ms,0,blend_radius_m)
    |   movel([0.353786, -1.256763, -2.648909, -0.806717, 1.570796, 1.924582],accel_mss,speed_ms,0,blend_radius_m)
    |   movel([0.355614, -1.255074, -2.649822, -0.807494, 1.570796, 1.926410],accel_mss,speed_ms,0,blend_radius_m)
    |   movel([0.355848, -1.254969, -2.649878, -0.807542, 1.570796, 1.926645],accel_mss,speed_ms,0,blend_radius_m)
    |   movel([0.356146, -1.255222, -2.649742, -0.807425, 1.570796, 1.926943],accel_mss,speed_ms,0,blend_radius_m)
    |   movel([0.356172, -1.255403, -2.649644, -0.807342, 1.570796, 1.926968],accel_mss,speed_ms,0,blend_radius_m)
    |   movel([0.355880, -1.255892, -2.649380, -0.807117, 1.570796, 1.926677],accel_mss,speed_ms,0,blend_radius_m)
    |   movel([0.355438, -1.256364, -2.649125, -0.806900, 1.570796, 1.926235],accel_mss,speed_ms,0,blend_radius_m)
    |   movel([0.354861, -1.257014, -2.648773, -0.806602, 1.570796, 1.925657],accel_mss,speed_ms,0,blend_radius_m)
    |   movel([0.354778, -1.257321, -2.648607, -0.806461, 1.570796, 1.925574],accel_mss,speed_ms,0,blend_radius_m)
    |   movel([0.355024, -1.257499, -2.648510, -0.806380, 1.570796, 1.925820],accel_mss,speed_ms,0,blend_radius_m)
    |   movel([0.355996, -1.257628, -2.648441, -0.806321, 1.570796, 1.926792],accel_mss,speed_ms,0,blend_radius_m)
    |   movel([0.357032, -1.257618, -2.648446, -0.806325, 1.570796, 1.927828],accel_mss,speed_ms,0,blend_radius_m)
    |   movel([0.358149, -1.257386, -2.648571, -0.806431, 1.570796, 1.928946],accel_mss,speed_ms,0,blend_radius_m)
    |   movel([0.359343, -1.256935, -2.648816, -0.806638, 1.570796, 1.930139],accel_mss,speed_ms,0,blend_radius_m)
    |   movel([0.360534, -1.256301, -2.649159, -0.806929, 1.570796, 1.931331],accel_mss,speed_ms,0,blend_radius_m)
    |   movel([0.361729, -1.255471, -2.649607, -0.807310, 1.570796, 1.932525],accel_mss,speed_ms,0,blend_radius_m)
    |   movel([0.362845, -1.254503, -2.650129, -0.807757, 1.570796, 1.933641],accel_mss,speed_ms,0,blend_radius_m)
    |   movel([0.363880, -1.253399, -2.650723, -0.808267, 1.570796, 1.934676],accel_mss,speed_ms,0,blend_radius_m)
    |   movel([0.364778, -1.252222, -2.651355, -0.808813, 1.570796, 1.935574],accel_mss,speed_ms,0,blend_radius_m)
    |   movel([0.365499, -1.251382, -2.651804, -0.809203, 1.570796, 1.936295],accel_mss,speed_ms,0,blend_radius_m)
    |   movel([0.365774, -1.251285, -2.651856, -0.809248, 1.570796, 1.936570],accel_mss,speed_ms,0,blend_radius_m)
    |   movel([0.366052, -1.251349, -2.651822, -0.809218, 1.570796, 1.936849],accel_mss,speed_ms,0,blend_radius_m)
    |   movel([0.366164, -1.251597, -2.651689, -0.809103, 1.570796, 1.936960],accel_mss,speed_ms,0,blend_radius_m)
    |   movel([0.366021, -1.252021, -2.651462, -0.808906, 1.570796, 1.936817],accel_mss,speed_ms,0,blend_radius_m)
    |   movel([0.365569, -1.252710, -2.651093, -0.808586, 1.570796, 1.936365],accel_mss,speed_ms,0,blend_radius_m)
    |   movel([0.364668, -1.253843, -2.650485, -0.808062, 1.570796, 1.935465],accel_mss,speed_ms,0,blend_radius_m)
    |   movel([0.363454, -1.255161, -2.649775, -0.807453, 1.570796, 1.934250],accel_mss,speed_ms,0,blend_radius_m)
    |   movel([0.362204, -1.256235, -2.649195, -0.806959, 1.570796, 1.933000],accel_mss,speed_ms,0,blend_radius_m)
    |   speed_ms = 0.005
    |   movel([0.362204, -1.246791, -2.644636, -0.820961, 1.570796, 1.933000],accel_mss,speed_ms,0,blend_radius_m)
    |   speed_ms = 0.040
    |   movel([0.376074, -1.237538, -2.649523, -0.825328, 1.570796, 1.946870],accel_mss,speed_ms,0,blend_radius_m)
    |   speed_ms = 0.005
    |   movel([0.376074, -1.247024, -2.654123, -0.811241, 1.570796, 1.946870],accel_mss,speed_ms,0,blend_radius_m)
    |   speed_ms = 0.025
    |   movel([0.376119, -1.247381, -2.653934, -0.811074, 1.570796, 1.946915],accel_mss,speed_ms,0,blend_radius_m)
    |   movel([0.375928, -1.247949, -2.653633, -0.810807, 1.570796, 1.946724],accel_mss,speed_ms,0,blend_radius_m)
    |   movel([0.375550, -1.248627, -2.653273, -0.810489, 1.570796, 1.946346],accel_mss,speed_ms,0,blend_radius_m)
    |   movel([0.374680, -1.249739, -2.652681, -0.809969, 1.570796, 1.945477],accel_mss,speed_ms,0,blend_radius_m)
    |   movel([0.374481, -1.250040, -2.652521, -0.809828, 1.570796, 1.945277],accel_mss,speed_ms,0,blend_radius_m)
    |   movel([0.374399, -1.250640, -2.652201, -0.809548, 1.570796, 1.945195],accel_mss,speed_ms,0,blend_radius_m)
    |   movel([0.374352, -1.250804, -2.652113, -0.809472, 1.570796, 1.945148],accel_mss,speed_ms,0,blend_radius_m)
    |   movel([0.373780, -1.251437, -2.651775, -0.809177, 1.570796, 1.944576],accel_mss,speed_ms,0,blend_radius_m)
    |   movel([0.373925, -1.250624, -2.652209, -0.809556, 1.570796, 1.944721],accel_mss,speed_ms,0,blend_radius_m)
    |   movel([0.373909, -1.250204, -2.652434, -0.809752, 1.570796, 1.944705],accel_mss,speed_ms,0,blend_radius_m)
    |   movel([0.373541, -1.249376, -2.652874, -0.810138, 1.570796, 1.944337],accel_mss,speed_ms,0,blend_radius_m)
    |   movel([0.372723, -1.248644, -2.653264, -0.810481, 1.570796, 1.943519],accel_mss,speed_ms,0,blend_radius_m)
    |   movel([0.371141, -1.247900, -2.653659, -0.810830, 1.570796, 1.941937],accel_mss,speed_ms,0,blend_radius_m)
    |   movel([0.370864, -1.247753, -2.653737, -0.810899, 1.570796, 1.941661],accel_mss,speed_ms,0,blend_radius_m)
    |   movel([0.370646, -1.247530, -2.653855, -0.811004, 1.570796, 1.941442],accel_mss,speed_ms,0,blend_radius_m)
    |   movel([0.370909, -1.247315, -2.653969, -0.811105, 1.570796, 1.941705],accel_mss,speed_ms,0,blend_radius_m)
    |   movel([0.373340, -1.247070, -2.654099, -0.811220, 1.570796, 1.944136],accel_mss,speed_ms,0,blend_radius_m)
    |   movel([0.375704, -1.246875, -2.654203, -0.811312, 1.570796, 1.946501],accel_mss,speed_ms,0,blend_radius_m)
    |   movel([0.376074, -1.247024, -2.654123, -0.811241, 1.570796, 1.946870],accel_mss,speed_ms,0,blend_radius_m)
    |   movel([0.376119, -1.247381, -2.653934, -0.811074, 1.570796, 1.946915],accel_mss,speed_ms,0,blend_radius_m)
    |   movel([0.375928, -1.247949, -2.653633, -0.810807, 1.570796, 1.946724],accel_mss,speed_ms,0,blend_radius_m)
    |   movel([0.375550, -1.248627, -2.653273, -0.810489, 1.570796, 1.946346],accel_mss,speed_ms,0,blend_radius_m)
    |   movel([0.374695, -1.249721, -2.652691, -0.809977, 1.570796, 1.945491],accel_mss,speed_ms,0,blend_radius_m)
    |   speed_ms = 0.005
    |   movel([0.374695, -1.240247, -2.648103, -0.824039, 1.570796, 1.945491],accel_mss,speed_ms,0,blend_radius_m)
    |   speed_ms = 0.040
    |   movel([0.390977, -1.218465, -2.659281, -0.834643, 1.570796, 1.961773],accel_mss,speed_ms,0,blend_radius_m)
    |   speed_ms = 0.005
    |   movel([0.390977, -1.228034, -2.663967, -0.820387, 1.570796, 1.961773],accel_mss,speed_ms,0,blend_radius_m)
    |   speed_ms = 0.025
    |   movel([0.390511, -1.229900, -2.663019, -0.819470, 1.570796, 1.961308],accel_mss,speed_ms,0,blend_radius_m)
    |   movel([0.389477, -1.232423, -2.661730, -0.818236, 1.570796, 1.960274],accel_mss,speed_ms,0,blend_radius_m)
    |   movel([0.388037, -1.235292, -2.660255, -0.816842, 1.570796, 1.958834],accel_mss,speed_ms,0,blend_radius_m)
    |   movel([0.386310, -1.238239, -2.658730, -0.815420, 1.570796, 1.957106],accel_mss,speed_ms,0,blend_radius_m)
    |   movel([0.382861, -1.243364, -2.656054, -0.812971, 1.570796, 1.953658],accel_mss,speed_ms,0,blend_radius_m)
    |   movel([0.380697, -1.246448, -2.654428, -0.811513, 1.570796, 1.951493],accel_mss,speed_ms,0,blend_radius_m)
    |   movel([0.378001, -1.249986, -2.652549, -0.809853, 1.570796, 1.948798],accel_mss,speed_ms,0,blend_radius_m)
    |   movel([0.376886, -1.251227, -2.651887, -0.809275, 1.570796, 1.947682],accel_mss,speed_ms,0,blend_radius_m)
    |   movel([0.375859, -1.252208, -2.651362, -0.808819, 1.570796, 1.946655],accel_mss,speed_ms,0,blend_radius_m)
    |   movel([0.374915, -1.252927, -2.650977, -0.808486, 1.570796, 1.945711],accel_mss,speed_ms,0,blend_radius_m)
    |   movel([0.373225, -1.253803, -2.650506, -0.808080, 1.570796, 1.944022],accel_mss,speed_ms,0,blend_radius_m)
    |   movel([0.372401, -1.254118, -2.650337, -0.807935, 1.570796, 1.943198],accel_mss,speed_ms,0,blend_radius_m)
    |   movel([0.372165, -1.254072, -2.650361, -0.807956, 1.570796, 1.942961],accel_mss,speed_ms,0,blend_radius_m)
    |   movel([0.374494, -1.252080, -2.651431, -0.808878, 1.570796, 1.945291],accel_mss,speed_ms,0,blend_radius_m)
    |   movel([0.375705, -1.250893, -2.652066, -0.809431, 1.570796, 1.946501],accel_mss,speed_ms,0,blend_radius_m)
    |   movel([0.379110, -1.247063, -2.654103, -0.811223, 1.570796, 1.949906],accel_mss,speed_ms,0,blend_radius_m)
    |   movel([0.382601, -1.242699, -2.656403, -0.813287, 1.570796, 1.953398],accel_mss,speed_ms,0,blend_radius_m)
    |   movel([0.385511, -1.238559, -2.658564, -0.815266, 1.570796, 1.956307],accel_mss,speed_ms,0,blend_radius_m)
    |   movel([0.386644, -1.236710, -2.659522, -0.816156, 1.570796, 1.957441],accel_mss,speed_ms,0,blend_radius_m)
    |   movel([0.387653, -1.234841, -2.660488, -0.817061, 1.570796, 1.958449],accel_mss,speed_ms,0,blend_radius_m)
    |   movel([0.388346, -1.233274, -2.661293, -0.817822, 1.570796, 1.959142],accel_mss,speed_ms,0,blend_radius_m)
    |   movel([0.388832, -1.231727, -2.662086, -0.818576, 1.570796, 1.959628],accel_mss,speed_ms,0,blend_radius_m)
    |   movel([0.389070, -1.230370, -2.662779, -0.819239, 1.570796, 1.959866],accel_mss,speed_ms,0,blend_radius_m)
    |   movel([0.389078, -1.229098, -2.663427, -0.819864, 1.570796, 1.959875],accel_mss,speed_ms,0,blend_radius_m)
    |   movel([0.388860, -1.227897, -2.664037, -0.820455, 1.570796, 1.959656],accel_mss,speed_ms,0,blend_radius_m)
    |   movel([0.388434, -1.226827, -2.664579, -0.820983, 1.570796, 1.959230],accel_mss,speed_ms,0,blend_radius_m)
    |   movel([0.387963, -1.225740, -2.665128, -0.821521, 1.570796, 1.958760],accel_mss,speed_ms,0,blend_radius_m)
    |   movel([0.387894, -1.224885, -2.665559, -0.821944, 1.570796, 1.958690],accel_mss,speed_ms,0,blend_radius_m)
    |   movel([0.388195, -1.223961, -2.666024, -0.822404, 1.570796, 1.958991],accel_mss,speed_ms,0,blend_radius_m)
    |   movel([0.389766, -1.221447, -2.667284, -0.823658, 1.570796, 1.960562],accel_mss,speed_ms,0,blend_radius_m)
    |   movel([0.389988, -1.221246, -2.667385, -0.823759, 1.570796, 1.960784],accel_mss,speed_ms,0,blend_radius_m)
    |   movel([0.389320, -1.222464, -2.666775, -0.823150, 1.570796, 1.960117],accel_mss,speed_ms,0,blend_radius_m)
    |   movel([0.388396, -1.224149, -2.665930, -0.822310, 1.570796, 1.959192],accel_mss,speed_ms,0,blend_radius_m)
    |   movel([0.388170, -1.224761, -2.665622, -0.822006, 1.570796, 1.958967],accel_mss,speed_ms,0,blend_radius_m)
    |   movel([0.388145, -1.225136, -2.665433, -0.821820, 1.570796, 1.958942],accel_mss,speed_ms,0,blend_radius_m)
    |   movel([0.388315, -1.225370, -2.665315, -0.821704, 1.570796, 1.959111],accel_mss,speed_ms,0,blend_radius_m)
    |   movel([0.388733, -1.225544, -2.665227, -0.821618, 1.570796, 1.959529],accel_mss,speed_ms,0,blend_radius_m)
    |   movel([0.389290, -1.225638, -2.665180, -0.821571, 1.570796, 1.960087],accel_mss,speed_ms,0,blend_radius_m)
    |   movel([0.390577, -1.225684, -2.665156, -0.821548, 1.570796, 1.961374],accel_mss,speed_ms,0,blend_radius_m)
    |   movel([0.390774, -1.225848, -2.665074, -0.821467, 1.570796, 1.961570],accel_mss,speed_ms,0,blend_radius_m)
    |   movel([0.391116, -1.226603, -2.664692, -0.821094, 1.570796, 1.961912],accel_mss,speed_ms,0,blend_radius_m)
    |   movel([0.391168, -1.226793, -2.664596, -0.821000, 1.570796, 1.961964],accel_mss,speed_ms,0,blend_radius_m)
    |   movel([0.390977, -1.228034, -2.663967, -0.820387, 1.570796, 1.961773],accel_mss,speed_ms,0,blend_radius_m)
    |   movel([0.390511, -1.229900, -2.663019, -0.819470, 1.570796, 1.961308],accel_mss,speed_ms,0,blend_radius_m)
    |   movel([0.390102, -1.230900, -2.662509, -0.818980, 1.570796, 1.960899],accel_mss,speed_ms,0,blend_radius_m)
    |   speed_ms = 0.005
    |   movel([0.390102, -1.221342, -2.657836, -0.833211, 1.570796, 1.960899],accel_mss,speed_ms,0,blend_radius_m)
    |   speed_ms = 0.040
    |   movel([0.371010, -1.233692, -2.651524, -0.827173, 1.570796, 1.941806],accel_mss,speed_ms,0,blend_radius_m)
    |   speed_ms = 0.005
    |   movel([0.371010, -1.243196, -2.656142, -0.813051, 1.570796, 1.941806],accel_mss,speed_ms,0,blend_radius_m)
    |   speed_ms = 0.025
    |   movel([0.371201, -1.243966, -2.655737, -0.812686, 1.570796, 1.941997],accel_mss,speed_ms,0,blend_radius_m)
    |   movel([0.371059, -1.244417, -2.655500, -0.812472, 1.570796, 1.941856],accel_mss,speed_ms,0,blend_radius_m)
    |   movel([0.370764, -1.244911, -2.655240, -0.812238, 1.570796, 1.941561],accel_mss,speed_ms,0,blend_radius_m)
    |   movel([0.370247, -1.245386, -2.654989, -0.812014, 1.570796, 1.941043],accel_mss,speed_ms,0,blend_radius_m)
    |   movel([0.369403, -1.245798, -2.654772, -0.811819, 1.570796, 1.940199],accel_mss,speed_ms,0,blend_radius_m)
    |   movel([0.368181, -1.246184, -2.654568, -0.811637, 1.570796, 1.938977],accel_mss,speed_ms,0,blend_radius_m)
    |   movel([0.363958, -1.247162, -2.654051, -0.811177, 1.570796, 1.934754],accel_mss,speed_ms,0,blend_radius_m)
    |   movel([0.363143, -1.247481, -2.653881, -0.811026, 1.570796, 1.933939],accel_mss,speed_ms,0,blend_radius_m)
    |   movel([0.361248, -1.248484, -2.653349, -0.810556, 1.570796, 1.932044],accel_mss,speed_ms,0,blend_radius_m)
    |   movel([0.360168, -1.249183, -2.652977, -0.810229, 1.570796, 1.930964],accel_mss,speed_ms,0,blend_radius_m)
    |   movel([0.356338, -1.251970, -2.651490, -0.808929, 1.570796, 1.927134],accel_mss,speed_ms,0,blend_radius_m)
    |   movel([0.355165, -1.252781, -2.651055, -0.808553, 1.570796, 1.925961],accel_mss,speed_ms,0,blend_radius_m)
    |   movel([0.353023, -1.254043, -2.650377, -0.807969, 1.570796, 1.923820],accel_mss,speed_ms,0,blend_radius_m)
    |   movel([0.351052, -1.255179, -2.649765, -0.807445, 1.570796, 1.921848],accel_mss,speed_ms,0,blend_radius_m)
    |   movel([0.349630, -1.256275, -2.649173, -0.806941, 1.570796, 1.920427],accel_mss,speed_ms,0,blend_radius_m)
    |   movel([0.348434, -1.257594, -2.648459, -0.806336, 1.570796, 1.919230],accel_mss,speed_ms,0,blend_radius_m)
    |   movel([0.346967, -1.259748, -2.647288, -0.805353, 1.570796, 1.917763],accel_mss,speed_ms,0,blend_radius_m)
    |   movel([0.347286, -1.258571, -2.647929, -0.805890, 1.570796, 1.918083],accel_mss,speed_ms,0,blend_radius_m)
    |   movel([0.348117, -1.256756, -2.648913, -0.806720, 1.570796, 1.918913],accel_mss,speed_ms,0,blend_radius_m)
    |   movel([0.348601, -1.256033, -2.649304, -0.807052, 1.570796, 1.919398],accel_mss,speed_ms,0,blend_radius_m)
    |   movel([0.349209, -1.255355, -2.649670, -0.807364, 1.570796, 1.920005],accel_mss,speed_ms,0,blend_radius_m)
    |   movel([0.350003, -1.254656, -2.650047, -0.807686, 1.570796, 1.920799],accel_mss,speed_ms,0,blend_radius_m)
    |   movel([0.350855, -1.254054, -2.650371, -0.807964, 1.570796, 1.921651],accel_mss,speed_ms,0,blend_radius_m)
    |   movel([0.353539, -1.252484, -2.651214, -0.808691, 1.570796, 1.924335],accel_mss,speed_ms,0,blend_radius_m)
    |   movel([0.355186, -1.251526, -2.651727, -0.809136, 1.570796, 1.925982],accel_mss,speed_ms,0,blend_radius_m)
    |   movel([0.356320, -1.250694, -2.652172, -0.809523, 1.570796, 1.927117],accel_mss,speed_ms,0,blend_radius_m)
    |   movel([0.357407, -1.249631, -2.652739, -0.810019, 1.570796, 1.928203],accel_mss,speed_ms,0,blend_radius_m)
    |   movel([0.358941, -1.247845, -2.653688, -0.810856, 1.570796, 1.929738],accel_mss,speed_ms,0,blend_radius_m)
    |   movel([0.361052, -1.245438, -2.654962, -0.811989, 1.570796, 1.931848],accel_mss,speed_ms,0,blend_radius_m)
    |   movel([0.362762, -1.243831, -2.655808, -0.812750, 1.570796, 1.933558],accel_mss,speed_ms,0,blend_radius_m)
    |   movel([0.364351, -1.242758, -2.656372, -0.813259, 1.570796, 1.935147],accel_mss,speed_ms,0,blend_radius_m)
    |   movel([0.366055, -1.242031, -2.656753, -0.813605, 1.570796, 1.936851],accel_mss,speed_ms,0,blend_radius_m)
    |   movel([0.367471, -1.241788, -2.656880, -0.813721, 1.570796, 1.938267],accel_mss,speed_ms,0,blend_radius_m)
    |   movel([0.368902, -1.241931, -2.656805, -0.813653, 1.570796, 1.939698],accel_mss,speed_ms,0,blend_radius_m)
    |   movel([0.370144, -1.242418, -2.656550, -0.813421, 1.570796, 1.940940],accel_mss,speed_ms,0,blend_radius_m)
    |   movel([0.371010, -1.243196, -2.656142, -0.813051, 1.570796, 1.941806],accel_mss,speed_ms,0,blend_radius_m)
    |   movel([0.371201, -1.243966, -2.655737, -0.812686, 1.570796, 1.941997],accel_mss,speed_ms,0,blend_radius_m)
    |   movel([0.371059, -1.244417, -2.655500, -0.812472, 1.570796, 1.941856],accel_mss,speed_ms,0,blend_radius_m)
    |   movel([0.370764, -1.244911, -2.655240, -0.812238, 1.570796, 1.941561],accel_mss,speed_ms,0,blend_radius_m)
    |   movel([0.370247, -1.245386, -2.654989, -0.812014, 1.570796, 1.941043],accel_mss,speed_ms,0,blend_radius_m)
    |   movel([0.369888, -1.245561, -2.654897, -0.811931, 1.570796, 1.940684],accel_mss,speed_ms,0,blend_radius_m)
    |   speed_ms = 0.005
    |   movel([0.369888, -1.236067, -2.650290, -0.826031, 1.570796, 1.940684],accel_mss,speed_ms,0,blend_radius_m)
    |   speed_ms = 0.040
    |   movel([0.362578, -1.233087, -2.651838, -0.827464, 1.570796, 1.933374],accel_mss,speed_ms,0,blend_radius_m)
    |   speed_ms = 0.005
    |   movel([0.362578, -1.242594, -2.656458, -0.813337, 1.570796, 1.933374],accel_mss,speed_ms,0,blend_radius_m)
    |   speed_ms = 0.025
    |   movel([0.361038, -1.243710, -2.655872, -0.812807, 1.570796, 1.931834],accel_mss,speed_ms,0,blend_radius_m)
    |   movel([0.359996, -1.244636, -2.655385, -0.812368, 1.570796, 1.930792],accel_mss,speed_ms,0,blend_radius_m)
    |   movel([0.356783, -1.247630, -2.653802, -0.810957, 1.570796, 1.927579],accel_mss,speed_ms,0,blend_radius_m)
    |   movel([0.354752, -1.249377, -2.652874, -0.810138, 1.570796, 1.925548],accel_mss,speed_ms,0,blend_radius_m)
    |   movel([0.347600, -1.255036, -2.649842, -0.807511, 1.570796, 1.918397],accel_mss,speed_ms,0,blend_radius_m)
    |   movel([0.346133, -1.257342, -2.648596, -0.806452, 1.570796, 1.916929],accel_mss,speed_ms,0,blend_radius_m)
    |   movel([0.342624, -1.262864, -2.645584, -0.803941, 1.570796, 1.913421],accel_mss,speed_ms,0,blend_radius_m)
    |   movel([0.342207, -1.263440, -2.645268, -0.803681, 1.570796, 1.913003],accel_mss,speed_ms,0,blend_radius_m)
    |   movel([0.341906, -1.263745, -2.645100, -0.803543, 1.570796, 1.912703],accel_mss,speed_ms,0,blend_radius_m)
    |   movel([0.341644, -1.263870, -2.645031, -0.803487, 1.570796, 1.912440],accel_mss,speed_ms,0,blend_radius_m)
    |   movel([0.341356, -1.263765, -2.645089, -0.803535, 1.570796, 1.912152],accel_mss,speed_ms,0,blend_radius_m)
    |   movel([0.341334, -1.263427, -2.645275, -0.803687, 1.570796, 1.912131],accel_mss,speed_ms,0,blend_radius_m)
    |   movel([0.341654, -1.262713, -2.645667, -0.804009, 1.570796, 1.912450],accel_mss,speed_ms,0,blend_radius_m)
    |   movel([0.342482, -1.261309, -2.646436, -0.804644, 1.570796, 1.913278],accel_mss,speed_ms,0,blend_radius_m)
    |   movel([0.343588, -1.259292, -2.647536, -0.805561, 1.570796, 1.914384],accel_mss,speed_ms,0,blend_radius_m)
    |   movel([0.343562, -1.259150, -2.647613, -0.805625, 1.570796, 1.914358],accel_mss,speed_ms,0,blend_radius_m)
    |   movel([0.343543, -1.258549, -2.647941, -0.805900, 1.570796, 1.914339],accel_mss,speed_ms,0,blend_radius_m)
    |   movel([0.343619, -1.258230, -2.648114, -0.806045, 1.570796, 1.914415],accel_mss,speed_ms,0,blend_radius_m)
    |   movel([0.343847, -1.257416, -2.648555, -0.806418, 1.570796, 1.914644],accel_mss,speed_ms,0,blend_radius_m)
    |   movel([0.341977, -1.258939, -2.647729, -0.805722, 1.570796, 1.912773],accel_mss,speed_ms,0,blend_radius_m)
    |   movel([0.340112, -1.260459, -2.646900, -0.805030, 1.570796, 1.910908],accel_mss,speed_ms,0,blend_radius_m)
    |   movel([0.340818, -1.261056, -2.646574, -0.804759, 1.570796, 1.911614],accel_mss,speed_ms,0,blend_radius_m)
    |   movel([0.341521, -1.261652, -2.646248, -0.804489, 1.570796, 1.912317],accel_mss,speed_ms,0,blend_radius_m)
    |   movel([0.340964, -1.262292, -2.645898, -0.804199, 1.570796, 1.911760],accel_mss,speed_ms,0,blend_radius_m)
    |   movel([0.340436, -1.262800, -2.645619, -0.803970, 1.570796, 1.911232],accel_mss,speed_ms,0,blend_radius_m)
    |   movel([0.338957, -1.263977, -2.644973, -0.803439, 1.570796, 1.909754],accel_mss,speed_ms,0,blend_radius_m)
    |   movel([0.337470, -1.265124, -2.644341, -0.802924, 1.570796, 1.908267],accel_mss,speed_ms,0,blend_radius_m)
    |   movel([0.336853, -1.265515, -2.644125, -0.802749, 1.570796, 1.907650],accel_mss,speed_ms,0,blend_radius_m)
    |   movel([0.336831, -1.266299, -2.643692, -0.802398, 1.570796, 1.907628],accel_mss,speed_ms,0,blend_radius_m)
    |   movel([0.336867, -1.267052, -2.643275, -0.802061, 1.570796, 1.907663],accel_mss,speed_ms,0,blend_radius_m)
    |   movel([0.340517, -1.264779, -2.644531, -0.803079, 1.570796, 1.911313],accel_mss,speed_ms,0,blend_radius_m)
    |   movel([0.342403, -1.263733, -2.645107, -0.803549, 1.570796, 1.913199],accel_mss,speed_ms,0,blend_radius_m)
    |   movel([0.344152, -1.262830, -2.645603, -0.803956, 1.570796, 1.914948],accel_mss,speed_ms,0,blend_radius_m)
    |   movel([0.345214, -1.262384, -2.645848, -0.804158, 1.570796, 1.916011],accel_mss,speed_ms,0,blend_radius_m)
    |   movel([0.345685, -1.262168, -2.645966, -0.804255, 1.570796, 1.916481],accel_mss,speed_ms,0,blend_radius_m)
    |   movel([0.345501, -1.261515, -2.646323, -0.804551, 1.570796, 1.916297],accel_mss,speed_ms,0,blend_radius_m)
    |   movel([0.345506, -1.261062, -2.646571, -0.804756, 1.570796, 1.916302],accel_mss,speed_ms,0,blend_radius_m)
    |   movel([0.345867, -1.259465, -2.647442, -0.805482, 1.570796, 1.916663],accel_mss,speed_ms,0,blend_radius_m)
    |   movel([0.346497, -1.257714, -2.648394, -0.806281, 1.570796, 1.917293],accel_mss,speed_ms,0,blend_radius_m)
    |   movel([0.347280, -1.256276, -2.649172, -0.806940, 1.570796, 1.918077],accel_mss,speed_ms,0,blend_radius_m)
    |   movel([0.348226, -1.255120, -2.649797, -0.807472, 1.570796, 1.919022],accel_mss,speed_ms,0,blend_radius_m)
    |   movel([0.349558, -1.253915, -2.650446, -0.808028, 1.570796, 1.920355],accel_mss,speed_ms,0,blend_radius_m)
    |   movel([0.351164, -1.252752, -2.651071, -0.808567, 1.570796, 1.921960],accel_mss,speed_ms,0,blend_radius_m)
    |   movel([0.354555, -1.250801, -2.652115, -0.809473, 1.570796, 1.925351],accel_mss,speed_ms,0,blend_radius_m)
    |   movel([0.355279, -1.250330, -2.652366, -0.809693, 1.570796, 1.926075],accel_mss,speed_ms,0,blend_radius_m)
    |   movel([0.356183, -1.249556, -2.652779, -0.810054, 1.570796, 1.926979],accel_mss,speed_ms,0,blend_radius_m)
    |   movel([0.356868, -1.248813, -2.653174, -0.810402, 1.570796, 1.927664],accel_mss,speed_ms,0,blend_radius_m)
    |   movel([0.360083, -1.245105, -2.655137, -0.812146, 1.570796, 1.930879],accel_mss,speed_ms,0,blend_radius_m)
    |   movel([0.360925, -1.244233, -2.655597, -0.812559, 1.570796, 1.931721],accel_mss,speed_ms,0,blend_radius_m)
    |   movel([0.362495, -1.242770, -2.656366, -0.813254, 1.570796, 1.933291],accel_mss,speed_ms,0,blend_radius_m)
    |   movel([0.362608, -1.242620, -2.656444, -0.813325, 1.570796, 1.933404],accel_mss,speed_ms,0,blend_radius_m)
    |   movel([0.361038, -1.243710, -2.655872, -0.812807, 1.570796, 1.931834],accel_mss,speed_ms,0,blend_radius_m)
    |   movel([0.359996, -1.244636, -2.655385, -0.812368, 1.570796, 1.930792],accel_mss,speed_ms,0,blend_radius_m)
    |   speed_ms = 0.005
    |   movel([0.359996, -1.235138, -2.650774, -0.826477, 1.570796, 1.930792],accel_mss,speed_ms,0,blend_radius_m)
    |   speed_ms = 0.040
    |   movel([0.356661, -1.236451, -2.650090, -0.825848, 1.570796, 1.927458],accel_mss,speed_ms,0,blend_radius_m)
    |   speed_ms = 0.005
    |   movel([0.356661, -1.245942, -2.654696, -0.811751, 1.570796, 1.927458],accel_mss,speed_ms,0,blend_radius_m)
    |   speed_ms = 0.025
    |   movel([0.356681, -1.246099, -2.654613, -0.811677, 1.570796, 1.927477],accel_mss,speed_ms,0,blend_radius_m)
    |   movel([0.356595, -1.246704, -2.654293, -0.811392, 1.570796, 1.927392],accel_mss,speed_ms,0,blend_radius_m)
    |   movel([0.356374, -1.246949, -2.654163, -0.811277, 1.570796, 1.927170],accel_mss,speed_ms,0,blend_radius_m)
    |   movel([0.352993, -1.249677, -2.652714, -0.809998, 1.570796, 1.923789],accel_mss,speed_ms,0,blend_radius_m)
    |   movel([0.349598, -1.252380, -2.651270, -0.808739, 1.570796, 1.920394],accel_mss,speed_ms,0,blend_radius_m)
    |   movel([0.349113, -1.252515, -2.651198, -0.808676, 1.570796, 1.919909],accel_mss,speed_ms,0,blend_radius_m)
    |   movel([0.348746, -1.252299, -2.651313, -0.808776, 1.570796, 1.919542],accel_mss,speed_ms,0,blend_radius_m)
    |   movel([0.347707, -1.251290, -2.651853, -0.809245, 1.570796, 1.918503],accel_mss,speed_ms,0,blend_radius_m)
    |   movel([0.347687, -1.251103, -2.651953, -0.809332, 1.570796, 1.918483],accel_mss,speed_ms,0,blend_radius_m)
    |   movel([0.348857, -1.248936, -2.653109, -0.810344, 1.570796, 1.919653],accel_mss,speed_ms,0,blend_radius_m)
    |   movel([0.349324, -1.248058, -2.653575, -0.810756, 1.570796, 1.920120],accel_mss,speed_ms,0,blend_radius_m)
    |   movel([0.350635, -1.245162, -2.655108, -0.812120, 1.570796, 1.921431],accel_mss,speed_ms,0,blend_radius_m)
    |   movel([0.351087, -1.243753, -2.655849, -0.812787, 1.570796, 1.921884],accel_mss,speed_ms,0,blend_radius_m)
    |   movel([0.351192, -1.242820, -2.656339, -0.813230, 1.570796, 1.921988],accel_mss,speed_ms,0,blend_radius_m)
    |   movel([0.350965, -1.242172, -2.656679, -0.813538, 1.570796, 1.921761],accel_mss,speed_ms,0,blend_radius_m)
    |   movel([0.350393, -1.241679, -2.656937, -0.813773, 1.570796, 1.921189],accel_mss,speed_ms,0,blend_radius_m)
    |   movel([0.349775, -1.241334, -2.657118, -0.813938, 1.570796, 1.920571],accel_mss,speed_ms,0,blend_radius_m)
    |   movel([0.351488, -1.240432, -2.657588, -0.814368, 1.570796, 1.922285],accel_mss,speed_ms,0,blend_radius_m)
    |   movel([0.353202, -1.239529, -2.658059, -0.814801, 1.570796, 1.923998],accel_mss,speed_ms,0,blend_radius_m)
    |   movel([0.353492, -1.240001, -2.657813, -0.814575, 1.570796, 1.924288],accel_mss,speed_ms,0,blend_radius_m)
    |   movel([0.353599, -1.240218, -2.657700, -0.814470, 1.570796, 1.924396],accel_mss,speed_ms,0,blend_radius_m)
    |   movel([0.353724, -1.240956, -2.657315, -0.814118, 1.570796, 1.924520],accel_mss,speed_ms,0,blend_radius_m)
    |   movel([0.353494, -1.241813, -2.656867, -0.813709, 1.570796, 1.924291],accel_mss,speed_ms,0,blend_radius_m)
    |   movel([0.352853, -1.243282, -2.656097, -0.813010, 1.570796, 1.923649],accel_mss,speed_ms,0,blend_radius_m)
    |   movel([0.352033, -1.244911, -2.655240, -0.812238, 1.570796, 1.922829],accel_mss,speed_ms,0,blend_radius_m)
    |   movel([0.350730, -1.247127, -2.654069, -0.811193, 1.570796, 1.921527],accel_mss,speed_ms,0,blend_radius_m)
    |   movel([0.350372, -1.247759, -2.653734, -0.810896, 1.570796, 1.921168],accel_mss,speed_ms,0,blend_radius_m)
    |   movel([0.350068, -1.248420, -2.653383, -0.810586, 1.570796, 1.920864],accel_mss,speed_ms,0,blend_radius_m)
    |   movel([0.350219, -1.248552, -2.653313, -0.810524, 1.570796, 1.921015],accel_mss,speed_ms,0,blend_radius_m)
    |   movel([0.350895, -1.248367, -2.653411, -0.810611, 1.570796, 1.921691],accel_mss,speed_ms,0,blend_radius_m)
    |   movel([0.351189, -1.248113, -2.653546, -0.810730, 1.570796, 1.921986],accel_mss,speed_ms,0,blend_radius_m)
    |   movel([0.351651, -1.247469, -2.653888, -0.811032, 1.570796, 1.922447],accel_mss,speed_ms,0,blend_radius_m)
    |   movel([0.352532, -1.245993, -2.654669, -0.811727, 1.570796, 1.923328],accel_mss,speed_ms,0,blend_radius_m)
    |   movel([0.353701, -1.243825, -2.655811, -0.812752, 1.570796, 1.924497],accel_mss,speed_ms,0,blend_radius_m)
    |   movel([0.353911, -1.243390, -2.656040, -0.812959, 1.570796, 1.924708],accel_mss,speed_ms,0,blend_radius_m)
    |   movel([0.354077, -1.243329, -2.656072, -0.812988, 1.570796, 1.924873],accel_mss,speed_ms,0,blend_radius_m)
    |   movel([0.354176, -1.243633, -2.655912, -0.812843, 1.570796, 1.924972],accel_mss,speed_ms,0,blend_radius_m)
    |   movel([0.354043, -1.246085, -2.654620, -0.811684, 1.570796, 1.924839],accel_mss,speed_ms,0,blend_radius_m)
    |   movel([0.353986, -1.246445, -2.654430, -0.811514, 1.570796, 1.924783],accel_mss,speed_ms,0,blend_radius_m)
    |   movel([0.353548, -1.247020, -2.654126, -0.811244, 1.570796, 1.924345],accel_mss,speed_ms,0,blend_radius_m)
    |   movel([0.352860, -1.247579, -2.653829, -0.810981, 1.570796, 1.923657],accel_mss,speed_ms,0,blend_radius_m)
    |   movel([0.349274, -1.250118, -2.652479, -0.809791, 1.570796, 1.920071],accel_mss,speed_ms,0,blend_radius_m)
    |   movel([0.348812, -1.250549, -2.652249, -0.809591, 1.570796, 1.919608],accel_mss,speed_ms,0,blend_radius_m)
    |   movel([0.348694, -1.250863, -2.652081, -0.809444, 1.570796, 1.919490],accel_mss,speed_ms,0,blend_radius_m)
    |   movel([0.348847, -1.251119, -2.651945, -0.809325, 1.570796, 1.919644],accel_mss,speed_ms,0,blend_radius_m)
    |   movel([0.349088, -1.251167, -2.651919, -0.809303, 1.570796, 1.919885],accel_mss,speed_ms,0,blend_radius_m)
    |   movel([0.349386, -1.251062, -2.651975, -0.809352, 1.570796, 1.920183],accel_mss,speed_ms,0,blend_radius_m)
    |   movel([0.350877, -1.250132, -2.652472, -0.809785, 1.570796, 1.921673],accel_mss,speed_ms,0,blend_radius_m)
    |   movel([0.352674, -1.248839, -2.653161, -0.810390, 1.570796, 1.923471],accel_mss,speed_ms,0,blend_radius_m)
    |   movel([0.356309, -1.245872, -2.654733, -0.811784, 1.570796, 1.927106],accel_mss,speed_ms,0,blend_radius_m)
    |   movel([0.356540, -1.245811, -2.654765, -0.811813, 1.570796, 1.927336],accel_mss,speed_ms,0,blend_radius_m)
    |   movel([0.356661, -1.245942, -2.654696, -0.811751, 1.570796, 1.927458],accel_mss,speed_ms,0,blend_radius_m)
    |   movel([0.356681, -1.246099, -2.654613, -0.811677, 1.570796, 1.927477],accel_mss,speed_ms,0,blend_radius_m)
    |   movel([0.356595, -1.246704, -2.654293, -0.811392, 1.570796, 1.927392],accel_mss,speed_ms,0,blend_radius_m)
    |   movel([0.356374, -1.246949, -2.654163, -0.811277, 1.570796, 1.927170],accel_mss,speed_ms,0,blend_radius_m)
    |   movel([0.354711, -1.248290, -2.653452, -0.810647, 1.570796, 1.925508],accel_mss,speed_ms,0,blend_radius_m)
    |   speed_ms = 0.005
    |   movel([0.354711, -1.238809, -2.648858, -0.824722, 1.570796, 1.925508],accel_mss,speed_ms,0,blend_radius_m)
    |   speed_ms = 0.040
    |   movel([0.360041, -1.232900, -2.651934, -0.827554, 1.570796, 1.930837],accel_mss,speed_ms,0,blend_radius_m)
    |   speed_ms = 0.005
    |   movel([0.360041, -1.242408, -2.656555, -0.813426, 1.570796, 1.930837],accel_mss,speed_ms,0,blend_radius_m)
    |   speed_ms = 0.025
    |   movel([0.360226, -1.242546, -2.656483, -0.813360, 1.570796, 1.931022],accel_mss,speed_ms,0,blend_radius_m)
    |   movel([0.360450, -1.242954, -2.656269, -0.813166, 1.570796, 1.931246],accel_mss,speed_ms,0,blend_radius_m)
    |   movel([0.360354, -1.243099, -2.656193, -0.813097, 1.570796, 1.931151],accel_mss,speed_ms,0,blend_radius_m)
    |   movel([0.357904, -1.245392, -2.654986, -0.812011, 1.570796, 1.928700],accel_mss,speed_ms,0,blend_radius_m)
    |   movel([0.358011, -1.244717, -2.655342, -0.812330, 1.570796, 1.928807],accel_mss,speed_ms,0,blend_radius_m)
    |   movel([0.358020, -1.243336, -2.656068, -0.812985, 1.570796, 1.928817],accel_mss,speed_ms,0,blend_radius_m)
    |   movel([0.357912, -1.242646, -2.656430, -0.813312, 1.570796, 1.928708],accel_mss,speed_ms,0,blend_radius_m)
    |   movel([0.357660, -1.241919, -2.656811, -0.813658, 1.570796, 1.928457],accel_mss,speed_ms,0,blend_radius_m)
    |   movel([0.358412, -1.241830, -2.656858, -0.813701, 1.570796, 1.929208],accel_mss,speed_ms,0,blend_radius_m)
    |   movel([0.358971, -1.241947, -2.656797, -0.813645, 1.570796, 1.929768],accel_mss,speed_ms,0,blend_radius_m)
    |   movel([0.360041, -1.242408, -2.656555, -0.813426, 1.570796, 1.930837],accel_mss,speed_ms,0,blend_radius_m)
    |   movel([0.360226, -1.242546, -2.656483, -0.813360, 1.570796, 1.931022],accel_mss,speed_ms,0,blend_radius_m)
    |   movel([0.360450, -1.242954, -2.656269, -0.813166, 1.570796, 1.931246],accel_mss,speed_ms,0,blend_radius_m)
    |   movel([0.360354, -1.243099, -2.656193, -0.813097, 1.570796, 1.931151],accel_mss,speed_ms,0,blend_radius_m)
    |   movel([0.358742, -1.244607, -2.655400, -0.812382, 1.570796, 1.929538],accel_mss,speed_ms,0,blend_radius_m)
    |   speed_ms = 0.005
    |   movel([0.358742, -1.235109, -2.650789, -0.826491, 1.570796, 1.929538],accel_mss,speed_ms,0,blend_radius_m)
    |   speed_ms = 0.040
    |   movel([0.365982, -1.224860, -2.656056, -0.831473, 1.570796, 1.936779],accel_mss,speed_ms,0,blend_radius_m)
    |   speed_ms = 0.005
    |   movel([0.365982, -1.234402, -2.660713, -0.817273, 1.570796, 1.936779],accel_mss,speed_ms,0,blend_radius_m)
    |   speed_ms = 0.025
    |   movel([0.367197, -1.232837, -2.661517, -0.818034, 1.570796, 1.937994],accel_mss,speed_ms,0,blend_radius_m)
    |   movel([0.367268, -1.232547, -2.661666, -0.818176, 1.570796, 1.938064],accel_mss,speed_ms,0,blend_radius_m)
    |   movel([0.366994, -1.232225, -2.661831, -0.818332, 1.570796, 1.937791],accel_mss,speed_ms,0,blend_radius_m)
    |   movel([0.366753, -1.232271, -2.661808, -0.818310, 1.570796, 1.937549],accel_mss,speed_ms,0,blend_radius_m)
    |   movel([0.364453, -1.233584, -2.661134, -0.817671, 1.570796, 1.935249],accel_mss,speed_ms,0,blend_radius_m)
    |   movel([0.364762, -1.232675, -2.661601, -0.818113, 1.570796, 1.935559],accel_mss,speed_ms,0,blend_radius_m)
    |   movel([0.365018, -1.232150, -2.661870, -0.818370, 1.570796, 1.935815],accel_mss,speed_ms,0,blend_radius_m)
    |   movel([0.365981, -1.229715, -2.663113, -0.819561, 1.570796, 1.936778],accel_mss,speed_ms,0,blend_radius_m)
    |   movel([0.366249, -1.228652, -2.663654, -0.820083, 1.570796, 1.937045],accel_mss,speed_ms,0,blend_radius_m)
    |   movel([0.366169, -1.228250, -2.663858, -0.820281, 1.570796, 1.936966],accel_mss,speed_ms,0,blend_radius_m)
    |   movel([0.365894, -1.228176, -2.663896, -0.820318, 1.570796, 1.936690],accel_mss,speed_ms,0,blend_radius_m)
    |   movel([0.365535, -1.228339, -2.663813, -0.820237, 1.570796, 1.936331],accel_mss,speed_ms,0,blend_radius_m)
    |   movel([0.365029, -1.228820, -2.663568, -0.820000, 1.570796, 1.935826],accel_mss,speed_ms,0,blend_radius_m)
    |   movel([0.363201, -1.231093, -2.662410, -0.818886, 1.570796, 1.933998],accel_mss,speed_ms,0,blend_radius_m)
    |   movel([0.363614, -1.229594, -2.663175, -0.819620, 1.570796, 1.934410],accel_mss,speed_ms,0,blend_radius_m)
    |   movel([0.364118, -1.227284, -2.664348, -0.820757, 1.570796, 1.934914],accel_mss,speed_ms,0,blend_radius_m)
    |   movel([0.364065, -1.226690, -2.664649, -0.821051, 1.570796, 1.934862],accel_mss,speed_ms,0,blend_radius_m)
    |   movel([0.363739, -1.226588, -2.664700, -0.821101, 1.570796, 1.934536],accel_mss,speed_ms,0,blend_radius_m)
    |   movel([0.363146, -1.226966, -2.664509, -0.820914, 1.570796, 1.933942],accel_mss,speed_ms,0,blend_radius_m)
    |   movel([0.362214, -1.227945, -2.664013, -0.820431, 1.570796, 1.933010],accel_mss,speed_ms,0,blend_radius_m)
    |   movel([0.361784, -1.228421, -2.663771, -0.820197, 1.570796, 1.932580],accel_mss,speed_ms,0,blend_radius_m)
    |   movel([0.360933, -1.229255, -2.663347, -0.819787, 1.570796, 1.931729],accel_mss,speed_ms,0,blend_radius_m)
    |   movel([0.360898, -1.228566, -2.663697, -0.820125, 1.570796, 1.931694],accel_mss,speed_ms,0,blend_radius_m)
    |   movel([0.360986, -1.227714, -2.664130, -0.820545, 1.570796, 1.931782],accel_mss,speed_ms,0,blend_radius_m)
    |   movel([0.360915, -1.226464, -2.664763, -0.821163, 1.570796, 1.931712],accel_mss,speed_ms,0,blend_radius_m)
    |   movel([0.360763, -1.225272, -2.665364, -0.821753, 1.570796, 1.931560],accel_mss,speed_ms,0,blend_radius_m)
    |   movel([0.360542, -1.224807, -2.665599, -0.821983, 1.570796, 1.931338],accel_mss,speed_ms,0,blend_radius_m)
    |   movel([0.360277, -1.224674, -2.665666, -0.822049, 1.570796, 1.931074],accel_mss,speed_ms,0,blend_radius_m)
    |   movel([0.359953, -1.224744, -2.665630, -0.822015, 1.570796, 1.930749],accel_mss,speed_ms,0,blend_radius_m)
    |   movel([0.359649, -1.225001, -2.665501, -0.821887, 1.570796, 1.930445],accel_mss,speed_ms,0,blend_radius_m)
    |   movel([0.359208, -1.225863, -2.665066, -0.821460, 1.570796, 1.930005],accel_mss,speed_ms,0,blend_radius_m)
    |   movel([0.358984, -1.226020, -2.664987, -0.821382, 1.570796, 1.929781],accel_mss,speed_ms,0,blend_radius_m)
    |   movel([0.358726, -1.225937, -2.665029, -0.821423, 1.570796, 1.929523],accel_mss,speed_ms,0,blend_radius_m)
    |   movel([0.358350, -1.225474, -2.665263, -0.821653, 1.570796, 1.929146],accel_mss,speed_ms,0,blend_radius_m)
    |   movel([0.357250, -1.224502, -2.665752, -0.822135, 1.570796, 1.928047],accel_mss,speed_ms,0,blend_radius_m)
    |   movel([0.356640, -1.224240, -2.665884, -0.822265, 1.570796, 1.927437],accel_mss,speed_ms,0,blend_radius_m)
    |   movel([0.356222, -1.224293, -2.665857, -0.822239, 1.570796, 1.927018],accel_mss,speed_ms,0,blend_radius_m)
    |   movel([0.355916, -1.224549, -2.665729, -0.822112, 1.570796, 1.926713],accel_mss,speed_ms,0,blend_radius_m)
    |   movel([0.355775, -1.224896, -2.665554, -0.821939, 1.570796, 1.926571],accel_mss,speed_ms,0,blend_radius_m)
    |   movel([0.355850, -1.225256, -2.665372, -0.821761, 1.570796, 1.926647],accel_mss,speed_ms,0,blend_radius_m)
    |   movel([0.356129, -1.225517, -2.665241, -0.821631, 1.570796, 1.926925],accel_mss,speed_ms,0,blend_radius_m)
    |   movel([0.356903, -1.226081, -2.664956, -0.821352, 1.570796, 1.927700],accel_mss,speed_ms,0,blend_radius_m)
    |   movel([0.357405, -1.226779, -2.664603, -0.821006, 1.570796, 1.928201],accel_mss,speed_ms,0,blend_radius_m)
    |   movel([0.357642, -1.227648, -2.664163, -0.820578, 1.570796, 1.928439],accel_mss,speed_ms,0,blend_radius_m)
    |   movel([0.357659, -1.229375, -2.663286, -0.819728, 1.570796, 1.928455],accel_mss,speed_ms,0,blend_radius_m)
    |   movel([0.357785, -1.229455, -2.663245, -0.819688, 1.570796, 1.928582],accel_mss,speed_ms,0,blend_radius_m)
    |   movel([0.358270, -1.229326, -2.663311, -0.819752, 1.570796, 1.929066],accel_mss,speed_ms,0,blend_radius_m)
    |   movel([0.358494, -1.229145, -2.663403, -0.819841, 1.570796, 1.929291],accel_mss,speed_ms,0,blend_radius_m)
    |   movel([0.358994, -1.228407, -2.663778, -0.820204, 1.570796, 1.929790],accel_mss,speed_ms,0,blend_radius_m)
    |   movel([0.359202, -1.228056, -2.663956, -0.820377, 1.570796, 1.929998],accel_mss,speed_ms,0,blend_radius_m)
    |   movel([0.359643, -1.227480, -2.664248, -0.820660, 1.570796, 1.930439],accel_mss,speed_ms,0,blend_radius_m)
    |   movel([0.359829, -1.227656, -2.664159, -0.820574, 1.570796, 1.930625],accel_mss,speed_ms,0,blend_radius_m)
    |   movel([0.359625, -1.228997, -2.663478, -0.819913, 1.570796, 1.930422],accel_mss,speed_ms,0,blend_radius_m)
    |   movel([0.359295, -1.230506, -2.662710, -0.819173, 1.570796, 1.930092],accel_mss,speed_ms,0,blend_radius_m)
    |   movel([0.358337, -1.233565, -2.661144, -0.817680, 1.570796, 1.929133],accel_mss,speed_ms,0,blend_radius_m)
    |   movel([0.358357, -1.233810, -2.661018, -0.817561, 1.570796, 1.929153],accel_mss,speed_ms,0,blend_radius_m)
    |   movel([0.358513, -1.233912, -2.660966, -0.817512, 1.570796, 1.929309],accel_mss,speed_ms,0,blend_radius_m)
    |   movel([0.358845, -1.233837, -2.661004, -0.817548, 1.570796, 1.929641],accel_mss,speed_ms,0,blend_radius_m)
    |   movel([0.359148, -1.233598, -2.661127, -0.817664, 1.570796, 1.929945],accel_mss,speed_ms,0,blend_radius_m)
    |   movel([0.359439, -1.233154, -2.661355, -0.817880, 1.570796, 1.930235],accel_mss,speed_ms,0,blend_radius_m)
    |   movel([0.359943, -1.231979, -2.661957, -0.818453, 1.570796, 1.930739],accel_mss,speed_ms,0,blend_radius_m)
    |   movel([0.360202, -1.231555, -2.662174, -0.818660, 1.570796, 1.930999],accel_mss,speed_ms,0,blend_radius_m)
    |   movel([0.362151, -1.229440, -2.663253, -0.819696, 1.570796, 1.932948],accel_mss,speed_ms,0,blend_radius_m)
    |   movel([0.362527, -1.229097, -2.663428, -0.819865, 1.570796, 1.933323],accel_mss,speed_ms,0,blend_radius_m)
    |   movel([0.362599, -1.229179, -2.663386, -0.819824, 1.570796, 1.933395],accel_mss,speed_ms,0,blend_radius_m)
    |   movel([0.361761, -1.231448, -2.662229, -0.818712, 1.570796, 1.932557],accel_mss,speed_ms,0,blend_radius_m)
    |   movel([0.361213, -1.232772, -2.661551, -0.818066, 1.570796, 1.932010],accel_mss,speed_ms,0,blend_radius_m)
    |   movel([0.360934, -1.233752, -2.661048, -0.817589, 1.570796, 1.931731],accel_mss,speed_ms,0,blend_radius_m)
    |   movel([0.361033, -1.233900, -2.660972, -0.817517, 1.570796, 1.931829],accel_mss,speed_ms,0,blend_radius_m)
    |   movel([0.361319, -1.233856, -2.660994, -0.817538, 1.570796, 1.932115],accel_mss,speed_ms,0,blend_radius_m)
    |   movel([0.361755, -1.233579, -2.661137, -0.817673, 1.570796, 1.932551],accel_mss,speed_ms,0,blend_radius_m)
    |   movel([0.363471, -1.232047, -2.661922, -0.818419, 1.570796, 1.934268],accel_mss,speed_ms,0,blend_radius_m)
    |   movel([0.364428, -1.231140, -2.662386, -0.818863, 1.570796, 1.935224],accel_mss,speed_ms,0,blend_radius_m)
    |   movel([0.363957, -1.232087, -2.661902, -0.818400, 1.570796, 1.934753],accel_mss,speed_ms,0,blend_radius_m)
    |   movel([0.363718, -1.232539, -2.661670, -0.818180, 1.570796, 1.934515],accel_mss,speed_ms,0,blend_radius_m)
    |   movel([0.362017, -1.235415, -2.660191, -0.816782, 1.570796, 1.932814],accel_mss,speed_ms,0,blend_radius_m)
    |   movel([0.361965, -1.235658, -2.660066, -0.816665, 1.570796, 1.932762],accel_mss,speed_ms,0,blend_radius_m)
    |   movel([0.362163, -1.235969, -2.659906, -0.816514, 1.570796, 1.932960],accel_mss,speed_ms,0,blend_radius_m)
    |   movel([0.362340, -1.235975, -2.659902, -0.816511, 1.570796, 1.933136],accel_mss,speed_ms,0,blend_radius_m)
    |   movel([0.364072, -1.235107, -2.660351, -0.816932, 1.570796, 1.934868],accel_mss,speed_ms,0,blend_radius_m)
    |   movel([0.362546, -1.236711, -2.659522, -0.816156, 1.570796, 1.933342],accel_mss,speed_ms,0,blend_radius_m)
    |   movel([0.361564, -1.237698, -2.659011, -0.815680, 1.570796, 1.932361],accel_mss,speed_ms,0,blend_radius_m)
    |   movel([0.361116, -1.238316, -2.658690, -0.815383, 1.570796, 1.931913],accel_mss,speed_ms,0,blend_radius_m)
    |   movel([0.361139, -1.238600, -2.658542, -0.815246, 1.570796, 1.931936],accel_mss,speed_ms,0,blend_radius_m)
    |   movel([0.361515, -1.238634, -2.658525, -0.815230, 1.570796, 1.932312],accel_mss,speed_ms,0,blend_radius_m)
    |   movel([0.362138, -1.238294, -2.658701, -0.815393, 1.570796, 1.932935],accel_mss,speed_ms,0,blend_radius_m)
    |   movel([0.363370, -1.237185, -2.659277, -0.815927, 1.570796, 1.934167],accel_mss,speed_ms,0,blend_radius_m)
    |   movel([0.364728, -1.235820, -2.659982, -0.816586, 1.570796, 1.935524],accel_mss,speed_ms,0,blend_radius_m)
    |   movel([0.365982, -1.234402, -2.660713, -0.817273, 1.570796, 1.936779],accel_mss,speed_ms,0,blend_radius_m)
    |   movel([0.367197, -1.232837, -2.661517, -0.818034, 1.570796, 1.937994],accel_mss,speed_ms,0,blend_radius_m)
    |   movel([0.367268, -1.232547, -2.661666, -0.818176, 1.570796, 1.938064],accel_mss,speed_ms,0,blend_radius_m)
    |   movel([0.366994, -1.232225, -2.661831, -0.818332, 1.570796, 1.937791],accel_mss,speed_ms,0,blend_radius_m)
    |   movel([0.366753, -1.232271, -2.661808, -0.818310, 1.570796, 1.937549],accel_mss,speed_ms,0,blend_radius_m)
    |   movel([0.366600, -1.232358, -2.661763, -0.818268, 1.570796, 1.937396],accel_mss,speed_ms,0,blend_radius_m)
    |   speed_ms = 0.005
    |   movel([0.366600, -1.222807, -2.657096, -0.832486, 1.570796, 1.937396],accel_mss,speed_ms,0,blend_radius_m)
    |   speed_ms = 0.040
    |   movel([0.357642, -1.227260, -2.654833, -0.830296, 1.570796, 1.928439],accel_mss,speed_ms,0,blend_radius_m)
    |   speed_ms = 0.005
    |   movel([0.357642, -1.236793, -2.659480, -0.816117, 1.570796, 1.928439],accel_mss,speed_ms,0,blend_radius_m)
    |   speed_ms = 0.025
    |   movel([0.358290, -1.237984, -2.658862, -0.815542, 1.570796, 1.929087],accel_mss,speed_ms,0,blend_radius_m)
    |   movel([0.355794, -1.236947, -2.659400, -0.816042, 1.570796, 1.926591],accel_mss,speed_ms,0,blend_radius_m)
    |   movel([0.355603, -1.236777, -2.659488, -0.816124, 1.570796, 1.926399],accel_mss,speed_ms,0,blend_radius_m)
    |   movel([0.355835, -1.236613, -2.659573, -0.816203, 1.570796, 1.926632],accel_mss,speed_ms,0,blend_radius_m)
    |   movel([0.356789, -1.235911, -2.659935, -0.816542, 1.570796, 1.927585],accel_mss,speed_ms,0,blend_radius_m)
    |   movel([0.356991, -1.235891, -2.659946, -0.816552, 1.570796, 1.927787],accel_mss,speed_ms,0,blend_radius_m)
    |   movel([0.357642, -1.236793, -2.659480, -0.816117, 1.570796, 1.928439],accel_mss,speed_ms,0,blend_radius_m)
    |   movel([0.358290, -1.237984, -2.658862, -0.815542, 1.570796, 1.929087],accel_mss,speed_ms,0,blend_radius_m)
    |   movel([0.357483, -1.237647, -2.659037, -0.815705, 1.570796, 1.928280],accel_mss,speed_ms,0,blend_radius_m)
    |   speed_ms = 0.005
    |   movel([0.357483, -1.228119, -2.654394, -0.829876, 1.570796, 1.928280],accel_mss,speed_ms,0,blend_radius_m)
    |   speed_ms = 0.040
    |   movel([0.353511, -1.228211, -2.654347, -0.829831, 1.570796, 1.924307],accel_mss,speed_ms,0,blend_radius_m)
    |   speed_ms = 0.005
    |   movel([0.353511, -1.237739, -2.658990, -0.815661, 1.570796, 1.924307],accel_mss,speed_ms,0,blend_radius_m)
    |   speed_ms = 0.025
    |   movel([0.352418, -1.237785, -2.658966, -0.815638, 1.570796, 1.923214],accel_mss,speed_ms,0,blend_radius_m)
    |   movel([0.352057, -1.237897, -2.658907, -0.815584, 1.570796, 1.922854],accel_mss,speed_ms,0,blend_radius_m)
    |   movel([0.350746, -1.238521, -2.658584, -0.815284, 1.570796, 1.921543],accel_mss,speed_ms,0,blend_radius_m)
    |   movel([0.348793, -1.239695, -2.657973, -0.814721, 1.570796, 1.919589],accel_mss,speed_ms,0,blend_radius_m)
    |   movel([0.346765, -1.241037, -2.657273, -0.814079, 1.570796, 1.917561],accel_mss,speed_ms,0,blend_radius_m)
    |   movel([0.345115, -1.242273, -2.656626, -0.813490, 1.570796, 1.915912],accel_mss,speed_ms,0,blend_radius_m)
    |   movel([0.344398, -1.242854, -2.656322, -0.813214, 1.570796, 1.915194],accel_mss,speed_ms,0,blend_radius_m)
    |   movel([0.345068, -1.243941, -2.655751, -0.812698, 1.570796, 1.915864],accel_mss,speed_ms,0,blend_radius_m)
    |   movel([0.345937, -1.245558, -2.654899, -0.811932, 1.570796, 1.916733],accel_mss,speed_ms,0,blend_radius_m)
    |   movel([0.346442, -1.247006, -2.654133, -0.811250, 1.570796, 1.917238],accel_mss,speed_ms,0,blend_radius_m)
    |   movel([0.346602, -1.248241, -2.653478, -0.810670, 1.570796, 1.917399],accel_mss,speed_ms,0,blend_radius_m)
    |   movel([0.346542, -1.248694, -2.653237, -0.810457, 1.570796, 1.917338],accel_mss,speed_ms,0,blend_radius_m)
    |   movel([0.346351, -1.249172, -2.652983, -0.810234, 1.570796, 1.917147],accel_mss,speed_ms,0,blend_radius_m)
    |   movel([0.346036, -1.249598, -2.652756, -0.810034, 1.570796, 1.916832],accel_mss,speed_ms,0,blend_radius_m)
    |   movel([0.345689, -1.249801, -2.652648, -0.809940, 1.570796, 1.916486],accel_mss,speed_ms,0,blend_radius_m)
    |   movel([0.345290, -1.249776, -2.652662, -0.809952, 1.570796, 1.916086],accel_mss,speed_ms,0,blend_radius_m)
    |   movel([0.343633, -1.248775, -2.653194, -0.810419, 1.570796, 1.914429],accel_mss,speed_ms,0,blend_radius_m)
    |   movel([0.343148, -1.248607, -2.653284, -0.810498, 1.570796, 1.913945],accel_mss,speed_ms,0,blend_radius_m)
    |   movel([0.342549, -1.248644, -2.653264, -0.810481, 1.570796, 1.913345],accel_mss,speed_ms,0,blend_radius_m)
    |   movel([0.342237, -1.249867, -2.652613, -0.809909, 1.570796, 1.913034],accel_mss,speed_ms,0,blend_radius_m)
    |   movel([0.342202, -1.250171, -2.652451, -0.809767, 1.570796, 1.912998],accel_mss,speed_ms,0,blend_radius_m)
    |   movel([0.342195, -1.250701, -2.652168, -0.809520, 1.570796, 1.912991],accel_mss,speed_ms,0,blend_radius_m)
    |   movel([0.342352, -1.250837, -2.652095, -0.809456, 1.570796, 1.913149],accel_mss,speed_ms,0,blend_radius_m)
    |   movel([0.344613, -1.250756, -2.652139, -0.809494, 1.570796, 1.915409],accel_mss,speed_ms,0,blend_radius_m)
    |   movel([0.345312, -1.250716, -2.652160, -0.809513, 1.570796, 1.916108],accel_mss,speed_ms,0,blend_radius_m)
    |   movel([0.346590, -1.250613, -2.652215, -0.809561, 1.570796, 1.917386],accel_mss,speed_ms,0,blend_radius_m)
    |   movel([0.346814, -1.250485, -2.652283, -0.809620, 1.570796, 1.917611],accel_mss,speed_ms,0,blend_radius_m)
    |   movel([0.347447, -1.249507, -2.652805, -0.810077, 1.570796, 1.918244],accel_mss,speed_ms,0,blend_radius_m)
    |   movel([0.348215, -1.248066, -2.653571, -0.810752, 1.570796, 1.919011],accel_mss,speed_ms,0,blend_radius_m)
    |   movel([0.349689, -1.244867, -2.655263, -0.812259, 1.570796, 1.920485],accel_mss,speed_ms,0,blend_radius_m)
    |   movel([0.349922, -1.244105, -2.655664, -0.812620, 1.570796, 1.920718],accel_mss,speed_ms,0,blend_radius_m)
    |   movel([0.349944, -1.243473, -2.655997, -0.812920, 1.570796, 1.920741],accel_mss,speed_ms,0,blend_radius_m)
    |   movel([0.349757, -1.243026, -2.656231, -0.813132, 1.570796, 1.920553],accel_mss,speed_ms,0,blend_radius_m)
    |   movel([0.349385, -1.242818, -2.656341, -0.813231, 1.570796, 1.920182],accel_mss,speed_ms,0,blend_radius_m)
    |   movel([0.348873, -1.242863, -2.656317, -0.813209, 1.570796, 1.919669],accel_mss,speed_ms,0,blend_radius_m)
    |   movel([0.348328, -1.242948, -2.656272, -0.813169, 1.570796, 1.919124],accel_mss,speed_ms,0,blend_radius_m)
    |   movel([0.348136, -1.242897, -2.656299, -0.813193, 1.570796, 1.918933],accel_mss,speed_ms,0,blend_radius_m)
    |   movel([0.347648, -1.242642, -2.656433, -0.813314, 1.570796, 1.918445],accel_mss,speed_ms,0,blend_radius_m)
    |   movel([0.347379, -1.242751, -2.656376, -0.813263, 1.570796, 1.918175],accel_mss,speed_ms,0,blend_radius_m)
    |   movel([0.346141, -1.243420, -2.656024, -0.812945, 1.570796, 1.916937],accel_mss,speed_ms,0,blend_radius_m)
    |   movel([0.345663, -1.243532, -2.655965, -0.812891, 1.570796, 1.916460],accel_mss,speed_ms,0,blend_radius_m)
    |   movel([0.345433, -1.243404, -2.656033, -0.812952, 1.570796, 1.916229],accel_mss,speed_ms,0,blend_radius_m)
    |   movel([0.345439, -1.243079, -2.656204, -0.813107, 1.570796, 1.916235],accel_mss,speed_ms,0,blend_radius_m)
    |   movel([0.345760, -1.242690, -2.656408, -0.813292, 1.570796, 1.916556],accel_mss,speed_ms,0,blend_radius_m)
    |   movel([0.347342, -1.241703, -2.656925, -0.813762, 1.570796, 1.918139],accel_mss,speed_ms,0,blend_radius_m)
    |   movel([0.354241, -1.237858, -2.658928, -0.815603, 1.570796, 1.925037],accel_mss,speed_ms,0,blend_radius_m)
    |   movel([0.353511, -1.237739, -2.658990, -0.815661, 1.570796, 1.924307],accel_mss,speed_ms,0,blend_radius_m)
    |   movel([0.352418, -1.237785, -2.658966, -0.815638, 1.570796, 1.923214],accel_mss,speed_ms,0,blend_radius_m)
    |   movel([0.352057, -1.237897, -2.658907, -0.815584, 1.570796, 1.922854],accel_mss,speed_ms,0,blend_radius_m)
    |   movel([0.350746, -1.238521, -2.658584, -0.815284, 1.570796, 1.921543],accel_mss,speed_ms,0,blend_radius_m)
    |   speed_ms = 0.005
    |   movel([0.350746, -1.228996, -2.653945, -0.829448, 1.570796, 1.921543],accel_mss,speed_ms,0,blend_radius_m)
    |   speed_ms = 0.040
    |   movel([0.354643, -1.220848, -2.658085, -0.833457, 1.570796, 1.925440],accel_mss,speed_ms,0,blend_radius_m)
    |   speed_ms = 0.005
    |   movel([0.354643, -1.230407, -2.662760, -0.819221, 1.570796, 1.925440],accel_mss,speed_ms,0,blend_radius_m)
    |   speed_ms = 0.025
    |   movel([0.355015, -1.230187, -2.662873, -0.819329, 1.570796, 1.925812],accel_mss,speed_ms,0,blend_radius_m)
    |   movel([0.355320, -1.229708, -2.663117, -0.819564, 1.570796, 1.926116],accel_mss,speed_ms,0,blend_radius_m)
    |   movel([0.355502, -1.229031, -2.663461, -0.819897, 1.570796, 1.926298],accel_mss,speed_ms,0,blend_radius_m)
    |   movel([0.355515, -1.228288, -2.663839, -0.820263, 1.570796, 1.926311],accel_mss,speed_ms,0,blend_radius_m)
    |   movel([0.355072, -1.226841, -2.664572, -0.820976, 1.570796, 1.925868],accel_mss,speed_ms,0,blend_radius_m)
    |   movel([0.354059, -1.225686, -2.665156, -0.821548, 1.570796, 1.924855],accel_mss,speed_ms,0,blend_radius_m)
    |   movel([0.353010, -1.225331, -2.665335, -0.821724, 1.570796, 1.923806],accel_mss,speed_ms,0,blend_radius_m)
    |   movel([0.352611, -1.225480, -2.665260, -0.821650, 1.570796, 1.923407],accel_mss,speed_ms,0,blend_radius_m)
    |   movel([0.352327, -1.225852, -2.665072, -0.821465, 1.570796, 1.923124],accel_mss,speed_ms,0,blend_radius_m)
    |   movel([0.352326, -1.226021, -2.664986, -0.821381, 1.570796, 1.923122],accel_mss,speed_ms,0,blend_radius_m)
    |   movel([0.353004, -1.226778, -2.664604, -0.821007, 1.570796, 1.923801],accel_mss,speed_ms,0,blend_radius_m)
    |   movel([0.353553, -1.227300, -2.664340, -0.820749, 1.570796, 1.924349],accel_mss,speed_ms,0,blend_radius_m)
    |   movel([0.353945, -1.227954, -2.664008, -0.820427, 1.570796, 1.924742],accel_mss,speed_ms,0,blend_radius_m)
    |   movel([0.354176, -1.228742, -2.663608, -0.820039, 1.570796, 1.924972],accel_mss,speed_ms,0,blend_radius_m)
    |   movel([0.354272, -1.230028, -2.662954, -0.819407, 1.570796, 1.925069],accel_mss,speed_ms,0,blend_radius_m)
    |   movel([0.354342, -1.230259, -2.662836, -0.819294, 1.570796, 1.925139],accel_mss,speed_ms,0,blend_radius_m)
    |   movel([0.354643, -1.230407, -2.662760, -0.819221, 1.570796, 1.925440],accel_mss,speed_ms,0,blend_radius_m)
    |   movel([0.355015, -1.230187, -2.662873, -0.819329, 1.570796, 1.925812],accel_mss,speed_ms,0,blend_radius_m)
    |   movel([0.355320, -1.229708, -2.663117, -0.819564, 1.570796, 1.926116],accel_mss,speed_ms,0,blend_radius_m)
    |   movel([0.355502, -1.229031, -2.663461, -0.819897, 1.570796, 1.926298],accel_mss,speed_ms,0,blend_radius_m)
    |   movel([0.355515, -1.228288, -2.663839, -0.820263, 1.570796, 1.926311],accel_mss,speed_ms,0,blend_radius_m)
    |   movel([0.355387, -1.227872, -2.664050, -0.820467, 1.570796, 1.926183],accel_mss,speed_ms,0,blend_radius_m)
    |   speed_ms = 0.005
    |   movel([0.355387, -1.218302, -2.659362, -0.834724, 1.570796, 1.926183],accel_mss,speed_ms,0,blend_radius_m)
    |   speed_ms = 0.040
    |   movel([0.350856, -1.220747, -2.658135, -0.833507, 1.570796, 1.921652],accel_mss,speed_ms,0,blend_radius_m)
    |   speed_ms = 0.005
    |   movel([0.350856, -1.230307, -2.662812, -0.819271, 1.570796, 1.921652],accel_mss,speed_ms,0,blend_radius_m)
    |   speed_ms = 0.025
    |   movel([0.350600, -1.230391, -2.662769, -0.819229, 1.570796, 1.921396],accel_mss,speed_ms,0,blend_radius_m)
    |   movel([0.350382, -1.230324, -2.662803, -0.819262, 1.570796, 1.921178],accel_mss,speed_ms,0,blend_radius_m)
    |   movel([0.349134, -1.228387, -2.663788, -0.820214, 1.570796, 1.919931],accel_mss,speed_ms,0,blend_radius_m)
    |   movel([0.348521, -1.229951, -2.662993, -0.819445, 1.570796, 1.919317],accel_mss,speed_ms,0,blend_radius_m)
    |   movel([0.347909, -1.231511, -2.662197, -0.818681, 1.570796, 1.918706],accel_mss,speed_ms,0,blend_radius_m)
    |   movel([0.346169, -1.231689, -2.662106, -0.818595, 1.570796, 1.916965],accel_mss,speed_ms,0,blend_radius_m)
    |   movel([0.344444, -1.231930, -2.661982, -0.818476, 1.570796, 1.915240],accel_mss,speed_ms,0,blend_radius_m)
    |   movel([0.344640, -1.233534, -2.661160, -0.817695, 1.570796, 1.915436],accel_mss,speed_ms,0,blend_radius_m)
    |   movel([0.344681, -1.234431, -2.660699, -0.817259, 1.570796, 1.915477],accel_mss,speed_ms,0,blend_radius_m)
    |   movel([0.344637, -1.235249, -2.660277, -0.816863, 1.570796, 1.915433],accel_mss,speed_ms,0,blend_radius_m)
    |   movel([0.344470, -1.235594, -2.660099, -0.816696, 1.570796, 1.915266],accel_mss,speed_ms,0,blend_radius_m)
    |   movel([0.344089, -1.235819, -2.659983, -0.816587, 1.570796, 1.914885],accel_mss,speed_ms,0,blend_radius_m)
    |   movel([0.343762, -1.235723, -2.660033, -0.816634, 1.570796, 1.914558],accel_mss,speed_ms,0,blend_radius_m)
    |   movel([0.343492, -1.235179, -2.660313, -0.816897, 1.570796, 1.914289],accel_mss,speed_ms,0,blend_radius_m)
    |   movel([0.343273, -1.234117, -2.660860, -0.817412, 1.570796, 1.914069],accel_mss,speed_ms,0,blend_radius_m)
    |   movel([0.342832, -1.231819, -2.662039, -0.818531, 1.570796, 1.913629],accel_mss,speed_ms,0,blend_radius_m)
    |   movel([0.342850, -1.231605, -2.662149, -0.818635, 1.570796, 1.913647],accel_mss,speed_ms,0,blend_radius_m)
    |   movel([0.342999, -1.231219, -2.662346, -0.818824, 1.570796, 1.913795],accel_mss,speed_ms,0,blend_radius_m)
    |   movel([0.343227, -1.231005, -2.662455, -0.818929, 1.570796, 1.914023],accel_mss,speed_ms,0,blend_radius_m)
    |   movel([0.344089, -1.230767, -2.662577, -0.819045, 1.570796, 1.914886],accel_mss,speed_ms,0,blend_radius_m)
    |   movel([0.345244, -1.230648, -2.662638, -0.819104, 1.570796, 1.916040],accel_mss,speed_ms,0,blend_radius_m)
    |   movel([0.347224, -1.230464, -2.662731, -0.819194, 1.570796, 1.918021],accel_mss,speed_ms,0,blend_radius_m)
    |   movel([0.347611, -1.229407, -2.663270, -0.819712, 1.570796, 1.918407],accel_mss,speed_ms,0,blend_radius_m)
    |   movel([0.348475, -1.227254, -2.664363, -0.820772, 1.570796, 1.919271],accel_mss,speed_ms,0,blend_radius_m)
    |   movel([0.348738, -1.226877, -2.664554, -0.820958, 1.570796, 1.919534],accel_mss,speed_ms,0,blend_radius_m)
    |   movel([0.349123, -1.226605, -2.664692, -0.821093, 1.570796, 1.919919],accel_mss,speed_ms,0,blend_radius_m)
    |   movel([0.349504, -1.226524, -2.664732, -0.821133, 1.570796, 1.920301],accel_mss,speed_ms,0,blend_radius_m)
    |   movel([0.349773, -1.226655, -2.664666, -0.821068, 1.570796, 1.920570],accel_mss,speed_ms,0,blend_radius_m)
    |   movel([0.350665, -1.228005, -2.663982, -0.820402, 1.570796, 1.921461],accel_mss,speed_ms,0,blend_radius_m)
    |   movel([0.351462, -1.229684, -2.663129, -0.819576, 1.570796, 1.922258],accel_mss,speed_ms,0,blend_radius_m)
    |   movel([0.350856, -1.230307, -2.662812, -0.819271, 1.570796, 1.921652],accel_mss,speed_ms,0,blend_radius_m)
    |   movel([0.350600, -1.230391, -2.662769, -0.819229, 1.570796, 1.921396],accel_mss,speed_ms,0,blend_radius_m)
    |   movel([0.350382, -1.230324, -2.662803, -0.819262, 1.570796, 1.921178],accel_mss,speed_ms,0,blend_radius_m)
    |   movel([0.349410, -1.228816, -2.663571, -0.820003, 1.570796, 1.920207],accel_mss,speed_ms,0,blend_radius_m)
    |   speed_ms = 0.005
    |   movel([0.349410, -1.219250, -2.658888, -0.834252, 1.570796, 1.920207],accel_mss,speed_ms,0,blend_radius_m)
    |   speed_ms = 0.040
    |   movel([0.341648, -1.226856, -2.655040, -0.830494, 1.570796, 1.912445],accel_mss,speed_ms,0,blend_radius_m)
    |   speed_ms = 0.005
    |   movel([0.341648, -1.236390, -2.659688, -0.816311, 1.570796, 1.912445],accel_mss,speed_ms,0,blend_radius_m)
    |   speed_ms = 0.025
    |   movel([0.342042, -1.236236, -2.659767, -0.816385, 1.570796, 1.912838],accel_mss,speed_ms,0,blend_radius_m)
    |   movel([0.342168, -1.236074, -2.659851, -0.816464, 1.570796, 1.912964],accel_mss,speed_ms,0,blend_radius_m)
    |   movel([0.342331, -1.235560, -2.660117, -0.816712, 1.570796, 1.913128],accel_mss,speed_ms,0,blend_radius_m)
    |   movel([0.342273, -1.235397, -2.660201, -0.816791, 1.570796, 1.913070],accel_mss,speed_ms,0,blend_radius_m)
    |   movel([0.341321, -1.235166, -2.660320, -0.816903, 1.570796, 1.912117],accel_mss,speed_ms,0,blend_radius_m)
    |   movel([0.340896, -1.235096, -2.660356, -0.816937, 1.570796, 1.911692],accel_mss,speed_ms,0,blend_radius_m)
    |   movel([0.338945, -1.234844, -2.660486, -0.817059, 1.570796, 1.909742],accel_mss,speed_ms,0,blend_radius_m)
    |   movel([0.338509, -1.234921, -2.660446, -0.817022, 1.570796, 1.909305],accel_mss,speed_ms,0,blend_radius_m)
    |   movel([0.338254, -1.235086, -2.660361, -0.816942, 1.570796, 1.909050],accel_mss,speed_ms,0,blend_radius_m)
    |   movel([0.338143, -1.235290, -2.660256, -0.816843, 1.570796, 1.908939],accel_mss,speed_ms,0,blend_radius_m)
    |   movel([0.337238, -1.239690, -2.657976, -0.814724, 1.570796, 1.908034],accel_mss,speed_ms,0,blend_radius_m)
    |   movel([0.337295, -1.239971, -2.657829, -0.814589, 1.570796, 1.908091],accel_mss,speed_ms,0,blend_radius_m)
    |   movel([0.337551, -1.240078, -2.657774, -0.814538, 1.570796, 1.908348],accel_mss,speed_ms,0,blend_radius_m)
    |   movel([0.337900, -1.239963, -2.657833, -0.814593, 1.570796, 1.908697],accel_mss,speed_ms,0,blend_radius_m)
    |   movel([0.338314, -1.239460, -2.658095, -0.814834, 1.570796, 1.909111],accel_mss,speed_ms,0,blend_radius_m)
    |   movel([0.338472, -1.238982, -2.658344, -0.815063, 1.570796, 1.909268],accel_mss,speed_ms,0,blend_radius_m)
    |   movel([0.339165, -1.236218, -2.659777, -0.816394, 1.570796, 1.909962],accel_mss,speed_ms,0,blend_radius_m)
    |   movel([0.341648, -1.236390, -2.659688, -0.816311, 1.570796, 1.912445],accel_mss,speed_ms,0,blend_radius_m)
    |   movel([0.342042, -1.236236, -2.659767, -0.816385, 1.570796, 1.912838],accel_mss,speed_ms,0,blend_radius_m)
    |   movel([0.342168, -1.236074, -2.659851, -0.816464, 1.570796, 1.912964],accel_mss,speed_ms,0,blend_radius_m)
    |   movel([0.342331, -1.235560, -2.660117, -0.816712, 1.570796, 1.913128],accel_mss,speed_ms,0,blend_radius_m)
    |   movel([0.342273, -1.235397, -2.660201, -0.816791, 1.570796, 1.913070],accel_mss,speed_ms,0,blend_radius_m)
    |   movel([0.341321, -1.235166, -2.660320, -0.816903, 1.570796, 1.912117],accel_mss,speed_ms,0,blend_radius_m)
    |   movel([0.340968, -1.235110, -2.660349, -0.816930, 1.570796, 1.911765],accel_mss,speed_ms,0,blend_radius_m)
    |   speed_ms = 0.005
    |   movel([0.340968, -1.225570, -2.655695, -0.831124, 1.570796, 1.911765],accel_mss,speed_ms,0,blend_radius_m)
    |   speed_ms = 0.040
    |   movel([0.335204, -1.206135, -2.665369, -0.840885, 1.570796, 1.906000],accel_mss,speed_ms,0,blend_radius_m)
    |   speed_ms = 0.005
    |   movel([0.335204, -1.215753, -2.670111, -0.826525, 1.570796, 1.906000],accel_mss,speed_ms,0,blend_radius_m)
    |   speed_ms = 0.025
    |   movel([0.334209, -1.216834, -2.669577, -0.825977, 1.570796, 1.905006],accel_mss,speed_ms,0,blend_radius_m)
    |   movel([0.332461, -1.219038, -2.668485, -0.824866, 1.570796, 1.903257],accel_mss,speed_ms,0,blend_radius_m)
    |   movel([0.330642, -1.221390, -2.667313, -0.823686, 1.570796, 1.901438],accel_mss,speed_ms,0,blend_radius_m)
    |   movel([0.330692, -1.221548, -2.667233, -0.823607, 1.570796, 1.901488],accel_mss,speed_ms,0,blend_radius_m)
    |   movel([0.332873, -1.218922, -2.668542, -0.824925, 1.570796, 1.903669],accel_mss,speed_ms,0,blend_radius_m)
    |   movel([0.335771, -1.215265, -2.670352, -0.826772, 1.570796, 1.906568],accel_mss,speed_ms,0,blend_radius_m)
    |   movel([0.335204, -1.215753, -2.670111, -0.826525, 1.570796, 1.906000],accel_mss,speed_ms,0,blend_radius_m)
    |   movel([0.334209, -1.216834, -2.669577, -0.825977, 1.570796, 1.905006],accel_mss,speed_ms,0,blend_radius_m)
    |   movel([0.332869, -1.218521, -2.668741, -0.825126, 1.570796, 1.903666],accel_mss,speed_ms,0,blend_radius_m)
    |   speed_ms = 0.005
    |   movel([0.332869, -1.208914, -2.664012, -0.839463, 1.570796, 1.903666],accel_mss,speed_ms,0,blend_radius_m)
    |   speed_ms = 0.040
    |   movel([0.328116, -1.227208, -2.654860, -0.830321, 1.570796, 1.898912],accel_mss,speed_ms,0,blend_radius_m)
    |   speed_ms = 0.005
    |   movel([0.328116, -1.236741, -2.659507, -0.816142, 1.570796, 1.898912],accel_mss,speed_ms,0,blend_radius_m)
    |   speed_ms = 0.025
    |   movel([0.328074, -1.235790, -2.659998, -0.816601, 1.570796, 1.898870],accel_mss,speed_ms,0,blend_radius_m)
    |   movel([0.327897, -1.235009, -2.660401, -0.816979, 1.570796, 1.898693],accel_mss,speed_ms,0,blend_radius_m)
    |   movel([0.326869, -1.233247, -2.661307, -0.817835, 1.570796, 1.897665],accel_mss,speed_ms,0,blend_radius_m)
    |   movel([0.326036, -1.231989, -2.661952, -0.818448, 1.570796, 1.896832],accel_mss,speed_ms,0,blend_radius_m)
    |   movel([0.325730, -1.231129, -2.662392, -0.818868, 1.570796, 1.896527],accel_mss,speed_ms,0,blend_radius_m)
    |   movel([0.325767, -1.230203, -2.662864, -0.819321, 1.570796, 1.896563],accel_mss,speed_ms,0,blend_radius_m)
    |   movel([0.326569, -1.227431, -2.664273, -0.820685, 1.570796, 1.897366],accel_mss,speed_ms,0,blend_radius_m)
    |   movel([0.325412, -1.229552, -2.663196, -0.819641, 1.570796, 1.896208],accel_mss,speed_ms,0,blend_radius_m)
    |   movel([0.325079, -1.231015, -2.662450, -0.818924, 1.570796, 1.895875],accel_mss,speed_ms,0,blend_radius_m)
    |   movel([0.325188, -1.232546, -2.661667, -0.818176, 1.570796, 1.895985],accel_mss,speed_ms,0,blend_radius_m)
    |   movel([0.325765, -1.234435, -2.660697, -0.817258, 1.570796, 1.896561],accel_mss,speed_ms,0,blend_radius_m)
    |   movel([0.326151, -1.235712, -2.660038, -0.816639, 1.570796, 1.896948],accel_mss,speed_ms,0,blend_radius_m)
    |   movel([0.326272, -1.236872, -2.659439, -0.816078, 1.570796, 1.897069],accel_mss,speed_ms,0,blend_radius_m)
    |   movel([0.326146, -1.238152, -2.658775, -0.815462, 1.570796, 1.896943],accel_mss,speed_ms,0,blend_radius_m)
    |   movel([0.325761, -1.239807, -2.657915, -0.814668, 1.570796, 1.896557],accel_mss,speed_ms,0,blend_radius_m)
    |   movel([0.324856, -1.242448, -2.656535, -0.813407, 1.570796, 1.895652],accel_mss,speed_ms,0,blend_radius_m)
    |   movel([0.323135, -1.246490, -2.654406, -0.811493, 1.570796, 1.893931],accel_mss,speed_ms,0,blend_radius_m)
    |   movel([0.321205, -1.250651, -2.652195, -0.809543, 1.570796, 1.892002],accel_mss,speed_ms,0,blend_radius_m)
    |   movel([0.319512, -1.253880, -2.650465, -0.808045, 1.570796, 1.890308],accel_mss,speed_ms,0,blend_radius_m)
    |   movel([0.318834, -1.255279, -2.649711, -0.807399, 1.570796, 1.889630],accel_mss,speed_ms,0,blend_radius_m)
    |   movel([0.323897, -1.246766, -2.654260, -0.811363, 1.570796, 1.894694],accel_mss,speed_ms,0,blend_radius_m)
    |   movel([0.325508, -1.243879, -2.655783, -0.812727, 1.570796, 1.896305],accel_mss,speed_ms,0,blend_radius_m)
    |   movel([0.326485, -1.241905, -2.656819, -0.813665, 1.570796, 1.897281],accel_mss,speed_ms,0,blend_radius_m)
    |   movel([0.327323, -1.239847, -2.657894, -0.814648, 1.570796, 1.898119],accel_mss,speed_ms,0,blend_radius_m)
    |   movel([0.327920, -1.238000, -2.658854, -0.815535, 1.570796, 1.898716],accel_mss,speed_ms,0,blend_radius_m)
    |   movel([0.328117, -1.236738, -2.659508, -0.816143, 1.570796, 1.898913],accel_mss,speed_ms,0,blend_radius_m)
    |   movel([0.328074, -1.235790, -2.659998, -0.816601, 1.570796, 1.898870],accel_mss,speed_ms,0,blend_radius_m)
